// TwinCAT 3 PLC project TSG_AmazonP_LM
// ProgramVersion: 3.1.4023.0
// libraries:
//   Lynus Energy Basic, * (Lynus AG)
//   Lynus Persistent Data V1, * (Lynus AG)
//   Lynus Standards, * (Lynus AG)
//   Tc2_ModbusSrv, * (Beckhoff Automation GmbH)
//   Tc2_Standard, * (Beckhoff Automation GmbH)
//   Tc2_System, * (Beckhoff Automation GmbH)
//   Tc2_Utilities, * (Beckhoff Automation GmbH)
//   Tc3_Module, * (Beckhoff Automation GmbH)
//   TSG Communicator, * (EfficientIO)
// project tree:
//   DUTs/ FB_ECS_Alfen_NG9xx_Platform.TcPOU, FB_ECS_Alpitronic_Hypercharger.TcPOU
//   / FastTask.TcTTO, PlcTask.TcTTO
//   POUs/ prgCS1.TcPOU, prgCS2.TcPOU, prgCS3.TcPOU, prgCS4.TcPOU, prgCS5.TcPOU, prgCS6.TcPOU, prgCS7.TcPOU, prgEM.TcPOU, prgEMS.TcPOU, prgLynusCom.TcPOU, prgLynusVar.TcPOU, prgPersData.TcPOU (not stored)
// real-time tasks:
//   TASK PlcTask: cycle T#10ms, priority 8, ADS port 350
//   TASK FastTask: cycle T#5ms, priority 6, ADS port 352
// I/O:
//   DEVICE Gerät 3 (CX-BK)
//     Box 1 (CX-BK)
// variable links:
//   TSG_AmazonP_LM/TSG_AmazonP_LM Instance <-> Device 3 (CX-BK)/Box 1 (CX-BK)
//     PlcTask Inputs/prgEM.fbEM1.fbKL3403.byStateCH1 <-> Term 2 (KL3403)/Channel 1/Status
//     PlcTask Inputs/prgEM.fbEM1.fbKL3403.byStateCH2 <-> Term 2 (KL3403)/Channel 2/Status
//     PlcTask Inputs/prgEM.fbEM1.fbKL3403.byStateCH3 <-> Term 2 (KL3403)/Channel 3/Status
//     PlcTask Inputs/prgEM.fbEM2.fbKL3403.byStateCH1 <-> Term 3 (KL3403)/Channel 1/Status
//     PlcTask Inputs/prgEM.fbEM2.fbKL3403.byStateCH2 <-> Term 3 (KL3403)/Channel 2/Status
//     PlcTask Inputs/prgEM.fbEM2.fbKL3403.byStateCH3 <-> Term 3 (KL3403)/Channel 3/Status
//     PlcTask Inputs/prgEM.fbEM3.fbKL3403.byStateCH1 <-> Term 4 (KL3403)/Channel 1/Status
//     PlcTask Inputs/prgEM.fbEM3.fbKL3403.byStateCH2 <-> Term 4 (KL3403)/Channel 2/Status
//     PlcTask Inputs/prgEM.fbEM3.fbKL3403.byStateCH3 <-> Term 4 (KL3403)/Channel 3/Status
//     PlcTask Inputs/prgEM.fbEM4.fbKL3403.byStateCH1 <-> Term 5 (KL3403)/Channel 1/Status
//     PlcTask Inputs/prgEM.fbEM4.fbKL3403.byStateCH2 <-> Term 5 (KL3403)/Channel 2/Status
//     PlcTask Inputs/prgEM.fbEM4.fbKL3403.byStateCH3 <-> Term 5 (KL3403)/Channel 3/Status
//     PlcTask Inputs/prgEM.fbEM5.fbKL3403.byStateCH1 <-> Term 6 (KL3403)/Channel 1/Status
//     PlcTask Inputs/prgEM.fbEM5.fbKL3403.byStateCH2 <-> Term 6 (KL3403)/Channel 2/Status
//     PlcTask Inputs/prgEM.fbEM5.fbKL3403.byStateCH3 <-> Term 6 (KL3403)/Channel 3/Status
//     PlcTask Inputs/prgEM.fbEM6.fbKL3403.byStateCH1 <-> Term 7 (KL3403)/Channel 1/Status
//     PlcTask Inputs/prgEM.fbEM6.fbKL3403.byStateCH2 <-> Term 7 (KL3403)/Channel 2/Status
//     PlcTask Inputs/prgEM.fbEM6.fbKL3403.byStateCH3 <-> Term 7 (KL3403)/Channel 3/Status
//     PlcTask Inputs/prgEM.fbEM7.fbKL3403.byStateCH1 <-> Term 8 (KL3403)/Channel 1/Status
//     PlcTask Inputs/prgEM.fbEM7.fbKL3403.byStateCH2 <-> Term 8 (KL3403)/Channel 2/Status
//     PlcTask Inputs/prgEM.fbEM7.fbKL3403.byStateCH3 <-> Term 8 (KL3403)/Channel 3/Status
//     PlcTask Inputs/prgEM.fbEM8.fbKL3403.byStateCH1 <-> Term 9 (KL3403)/Channel 1/Status
//     PlcTask Inputs/prgEM.fbEM8.fbKL3403.byStateCH2 <-> Term 9 (KL3403)/Channel 2/Status
//     PlcTask Inputs/prgEM.fbEM8.fbKL3403.byStateCH3 <-> Term 9 (KL3403)/Channel 3/Status
//     PlcTask Inputs/prgEM.fbEM1.fbKL3403.iDataInCH1 <-> Term 2 (KL3403)/Channel 1/Daten Ein
//     PlcTask Inputs/prgEM.fbEM1.fbKL3403.iDataInCH2 <-> Term 2 (KL3403)/Channel 2/Daten Ein
//     PlcTask Inputs/prgEM.fbEM1.fbKL3403.iDataInCH3 <-> Term 2 (KL3403)/Channel 3/Daten Ein
//     PlcTask Inputs/prgEM.fbEM2.fbKL3403.iDataInCH1 <-> Term 3 (KL3403)/Channel 1/Daten Ein
//     PlcTask Inputs/prgEM.fbEM2.fbKL3403.iDataInCH2 <-> Term 3 (KL3403)/Channel 2/Daten Ein
//     PlcTask Inputs/prgEM.fbEM2.fbKL3403.iDataInCH3 <-> Term 3 (KL3403)/Channel 3/Daten Ein
//     PlcTask Inputs/prgEM.fbEM3.fbKL3403.iDataInCH1 <-> Term 4 (KL3403)/Channel 1/Daten Ein
//     PlcTask Inputs/prgEM.fbEM3.fbKL3403.iDataInCH2 <-> Term 4 (KL3403)/Channel 2/Daten Ein
//     PlcTask Inputs/prgEM.fbEM3.fbKL3403.iDataInCH3 <-> Term 4 (KL3403)/Channel 3/Daten Ein
//     PlcTask Inputs/prgEM.fbEM4.fbKL3403.iDataInCH1 <-> Term 5 (KL3403)/Channel 1/Daten Ein
//     PlcTask Inputs/prgEM.fbEM4.fbKL3403.iDataInCH2 <-> Term 5 (KL3403)/Channel 2/Daten Ein
//     PlcTask Inputs/prgEM.fbEM4.fbKL3403.iDataInCH3 <-> Term 5 (KL3403)/Channel 3/Daten Ein
//     PlcTask Inputs/prgEM.fbEM5.fbKL3403.iDataInCH1 <-> Term 6 (KL3403)/Channel 1/Daten Ein
//     PlcTask Inputs/prgEM.fbEM5.fbKL3403.iDataInCH2 <-> Term 6 (KL3403)/Channel 2/Daten Ein
//     PlcTask Inputs/prgEM.fbEM5.fbKL3403.iDataInCH3 <-> Term 6 (KL3403)/Channel 3/Daten Ein
//     PlcTask Inputs/prgEM.fbEM6.fbKL3403.iDataInCH1 <-> Term 7 (KL3403)/Channel 1/Daten Ein
//     PlcTask Inputs/prgEM.fbEM6.fbKL3403.iDataInCH2 <-> Term 7 (KL3403)/Channel 2/Daten Ein
//     PlcTask Inputs/prgEM.fbEM6.fbKL3403.iDataInCH3 <-> Term 7 (KL3403)/Channel 3/Daten Ein
//     PlcTask Inputs/prgEM.fbEM7.fbKL3403.iDataInCH1 <-> Term 8 (KL3403)/Channel 1/Daten Ein
//     PlcTask Inputs/prgEM.fbEM7.fbKL3403.iDataInCH2 <-> Term 8 (KL3403)/Channel 2/Daten Ein
//     PlcTask Inputs/prgEM.fbEM7.fbKL3403.iDataInCH3 <-> Term 8 (KL3403)/Channel 3/Daten Ein
//     PlcTask Inputs/prgEM.fbEM8.fbKL3403.iDataInCH1 <-> Term 9 (KL3403)/Channel 1/Daten Ein
//     PlcTask Inputs/prgEM.fbEM8.fbKL3403.iDataInCH2 <-> Term 9 (KL3403)/Channel 2/Daten Ein
//     PlcTask Inputs/prgEM.fbEM8.fbKL3403.iDataInCH3 <-> Term 9 (KL3403)/Channel 3/Daten Ein
//     PlcTask Inputs/prgEM.fbKBusState.uiKBusState_OUT <-> Inputs/State
//     PlcTask Outputs/prgEM.fbEM1.fbKL3403.byCntrCH1 <-> Term 2 (KL3403)/Channel 1/Kontrolle
//     PlcTask Outputs/prgEM.fbEM1.fbKL3403.byCntrCH2 <-> Term 2 (KL3403)/Channel 2/Kontrolle
//     PlcTask Outputs/prgEM.fbEM1.fbKL3403.byCntrCH3 <-> Term 2 (KL3403)/Channel 3/Kontrolle
//     PlcTask Outputs/prgEM.fbEM2.fbKL3403.byCntrCH1 <-> Term 3 (KL3403)/Channel 1/Kontrolle
//     PlcTask Outputs/prgEM.fbEM2.fbKL3403.byCntrCH2 <-> Term 3 (KL3403)/Channel 2/Kontrolle
//     PlcTask Outputs/prgEM.fbEM2.fbKL3403.byCntrCH3 <-> Term 3 (KL3403)/Channel 3/Kontrolle
//     PlcTask Outputs/prgEM.fbEM3.fbKL3403.byCntrCH1 <-> Term 4 (KL3403)/Channel 1/Kontrolle
//     PlcTask Outputs/prgEM.fbEM3.fbKL3403.byCntrCH2 <-> Term 4 (KL3403)/Channel 2/Kontrolle
//     PlcTask Outputs/prgEM.fbEM3.fbKL3403.byCntrCH3 <-> Term 4 (KL3403)/Channel 3/Kontrolle
//     PlcTask Outputs/prgEM.fbEM4.fbKL3403.byCntrCH1 <-> Term 5 (KL3403)/Channel 1/Kontrolle
//     PlcTask Outputs/prgEM.fbEM4.fbKL3403.byCntrCH2 <-> Term 5 (KL3403)/Channel 2/Kontrolle
//     PlcTask Outputs/prgEM.fbEM4.fbKL3403.byCntrCH3 <-> Term 5 (KL3403)/Channel 3/Kontrolle
//     PlcTask Outputs/prgEM.fbEM5.fbKL3403.byCntrCH1 <-> Term 6 (KL3403)/Channel 1/Kontrolle
//     PlcTask Outputs/prgEM.fbEM5.fbKL3403.byCntrCH2 <-> Term 6 (KL3403)/Channel 2/Kontrolle
//     PlcTask Outputs/prgEM.fbEM5.fbKL3403.byCntrCH3 <-> Term 6 (KL3403)/Channel 3/Kontrolle
//     PlcTask Outputs/prgEM.fbEM6.fbKL3403.byCntrCH1 <-> Term 7 (KL3403)/Channel 1/Kontrolle
//     PlcTask Outputs/prgEM.fbEM6.fbKL3403.byCntrCH2 <-> Term 7 (KL3403)/Channel 2/Kontrolle
//     PlcTask Outputs/prgEM.fbEM6.fbKL3403.byCntrCH3 <-> Term 7 (KL3403)/Channel 3/Kontrolle
//     PlcTask Outputs/prgEM.fbEM7.fbKL3403.byCntrCH1 <-> Term 8 (KL3403)/Channel 1/Kontrolle
//     PlcTask Outputs/prgEM.fbEM7.fbKL3403.byCntrCH2 <-> Term 8 (KL3403)/Channel 2/Kontrolle
//     PlcTask Outputs/prgEM.fbEM7.fbKL3403.byCntrCH3 <-> Term 8 (KL3403)/Channel 3/Kontrolle
//     PlcTask Outputs/prgEM.fbEM8.fbKL3403.byCntrCH1 <-> Term 9 (KL3403)/Channel 1/Kontrolle
//     PlcTask Outputs/prgEM.fbEM8.fbKL3403.byCntrCH2 <-> Term 9 (KL3403)/Channel 2/Kontrolle
//     PlcTask Outputs/prgEM.fbEM8.fbKL3403.byCntrCH3 <-> Term 9 (KL3403)/Channel 3/Kontrolle

CONFIGURATION TSG_AmazonP_LM
    RESOURCE PLC ON TwinCAT3
        TASK FastTask(INTERVAL := T#5ms, PRIORITY := 6);
        TASK PlcTask(INTERVAL := T#10ms, PRIORITY := 8);
        PROGRAM prgLynusVar WITH FastTask : prgLynusVar;
        PROGRAM prgEMS WITH PlcTask : prgEMS;
        PROGRAM prgEM WITH PlcTask : prgEM;
        PROGRAM prgPersData WITH PlcTask : prgPersData;
        PROGRAM prgCS2 WITH PlcTask : prgCS2;
        PROGRAM prgCS3 WITH PlcTask : prgCS3;
        PROGRAM prgCS4 WITH PlcTask : prgCS4;
        PROGRAM prgCS5 WITH PlcTask : prgCS5;
        PROGRAM prgCS6 WITH PlcTask : prgCS6;
        PROGRAM prgCS7 WITH PlcTask : prgCS7;
        PROGRAM prgCS1 WITH PlcTask : prgCS1;
        PROGRAM prgLynusCom WITH PlcTask : prgLynusCom;
    END_RESOURCE
END_CONFIGURATION

// ---- POUs/prgLynusVar.TcPOU
PROGRAM prgLynusVar
VAR
	fbVarInfo			: FB_VarInfo;
	fbRW1				: FB_ReadWrite;
	fbRW2				: FB_ReadWrite;
	fbRW3				: FB_ReadWrite;
	fbRW4				: FB_ReadWrite;
	fbRW5				: FB_ReadWrite;
	fbRW6				: FB_ReadWrite;
	fbRW7				: FB_ReadWrite;
	fbRW8				: FB_ReadWrite;
	fbRW9				: FB_ReadWrite;
	fbRW10				: FB_ReadWrite;
	
	arrCount			: ARRAY[1..10] OF UDINT;
	arrSize				: ARRAY[1..10] OF UDINT;
	
	FPError				: ARRAY[1..10] OF R_TRIG;
	arrError			: ARRAY[1..10] OF UINT;
END_VAR

fbVarInfo(
	bReadInfo:= , 
	eTMCFile:= eSelectTMCFile.eUseTMCFile, 
	eSavePositionTMCFile:= eSavePositionOnPLC.ePostionC, 
	udiCounterFoundVariables=> , 
	bError=> , 
	bBusy=> , 
	byProgress=> , 
	udiErrorCodeOut=> , 
	eErrorVarInfo_Out=> , 
	sVarWithError=> );
	
fbRW1();
fbRW2();
fbRW3();
fbRW4();
fbRW5();
fbRW6();
fbRW7();
fbRW8();
fbRW9();
fbRW10();

FPError[1](CLK:= fbRW1.bError, Q=> );
FPError[2](CLK:= fbRW2.bError, Q=> );
FPError[3](CLK:= fbRW3.bError, Q=> );
FPError[4](CLK:= fbRW4.bError, Q=> );
FPError[5](CLK:= fbRW5.bError, Q=> );
FPError[6](CLK:= fbRW6.bError, Q=> );
FPError[7](CLK:= fbRW7.bError, Q=> );
FPError[8](CLK:= fbRW8.bError, Q=> );
FPError[9](CLK:= fbRW9.bError, Q=> );
FPError[10](CLK:= fbRW10.bError, Q=> );

IF FPError[1].Q THEN arrError[1] := arrError[1] + 1; END_IF 
IF FPError[2].Q THEN arrError[2] := arrError[2] + 1; END_IF 
IF FPError[3].Q THEN arrError[3] := arrError[3] + 1; END_IF 
IF FPError[4].Q THEN arrError[4] := arrError[4] + 1; END_IF 
IF FPError[5].Q THEN arrError[5] := arrError[5] + 1; END_IF 
IF FPError[6].Q THEN arrError[6] := arrError[6] + 1; END_IF 
IF FPError[7].Q THEN arrError[7] := arrError[7] + 1; END_IF 
IF FPError[8].Q THEN arrError[8] := arrError[8] + 1; END_IF 
IF FPError[9].Q THEN arrError[9] := arrError[9] + 1; END_IF 
IF FPError[10].Q THEN arrError[10] := arrError[10] + 1; END_IF

END_PROGRAM

// ---- POUs/prgEMS.TcPOU
PROGRAM prgEMS
VAR
	fbEMS		: FB_EMS_V2;		//{#lynus.ag#()}
	
	
	//Feedback CS
	arrTarget1			: ARRAY[1..12] OF REAL;
	arrTarget2			: ARRAY[1..10] OF REAL;
	arrTarget3			: ARRAY[1..10] OF REAL;
	arrTarget4			: ARRAY[1..10] OF REAL;
	arrTarget5			: ARRAY[1..10] OF REAL;
	arrTarget6			: ARRAY[1..10] OF REAL;
	arrTarget7			: ARRAY[1..2] OF REAL;
	
	arrPower1			: ARRAY[1..12] OF LREAL;
	arrPower2			: ARRAY[1..10] OF LREAL;
	arrPower3			: ARRAY[1..10] OF LREAL;
	arrPower4			: ARRAY[1..10] OF LREAL;
	arrPower5			: ARRAY[1..10] OF LREAL;
	arrPower6			: ARRAY[1..10] OF LREAL;
	arrPower7			: ARRAY[1..2] OF LREAL;
END_VAR

fbEMS(
	bEnable:= , 
	tDelayPwrCorrectionECS:= , 
	stNrOfEM_IN_ECS:= , 
	stSizeMainFuseCS:= , 
	stSetupEMS:= , 
	eOperationMode:= , 
	eSpeedModeBackendController:= E_SpeedModeBackendController_EMS.eSlow, 
	eSpeedModeLocalController:= E_SpeedModeLocalController_EMS.eSlow, 
	bActivateHP:= , 
	bControllingState:= , 
	rHeartbeat:= , 
	rErrorWarning:= , 
	rEnergyOptReady:= , 
	rNewBattPower:= , 
	eMessageEMS=> , 
	bStateEnable=> , 
	bStateAllowChrgFromGrid=> , 
	bMissingPowerData=> , 
	bSurplusAvailable=> , 
	bSEnableMainFuseFunc=> , 
	byProgress=> , 
	uiState_OUT=> , 
	diNrOfEMS_OUT=> , 
	arrMinPrioReached=> , 
	arrMaxPrioReached=> );
	
//Feedback
arrTarget1[1] := prgCS1.fbAlfen1.stDataECS.rTargetPower;
arrTarget1[2] := prgCS1.fbAlfen2.stDataECS.rTargetPower;
arrTarget1[3] := prgCS1.fbAlfen3.stDataECS.rTargetPower;
arrTarget1[4] := prgCS1.fbAlfen4.stDataECS.rTargetPower;
arrTarget1[5] := prgCS1.fbAlfen5.stDataECS.rTargetPower;
arrTarget1[6] := prgCS1.fbAlfen6.stDataECS.rTargetPower;
arrTarget1[7] := prgCS1.fbAlfen7.stDataECS.rTargetPower;
arrTarget1[8] := prgCS1.fbAlfen8.stDataECS.rTargetPower;
arrTarget1[9] := prgCS1.fbAlfen9.stDataECS.rTargetPower;
arrTarget1[10] := prgCS1.fbAlfen10.stDataECS.rTargetPower;
arrTarget1[11] := prgCS1.fbApliT_1.stDataECS.rTargetPower;
arrTarget1[12] := prgCS1.fbApliT_2.stDataECS.rTargetPower;

arrTarget2[1] := prgCS2.fbAlfen1.stDataECS.rTargetPower;
arrTarget2[2] := prgCS2.fbAlfen2.stDataECS.rTargetPower;
arrTarget2[3] := prgCS2.fbAlfen3.stDataECS.rTargetPower;
arrTarget2[4] := prgCS2.fbAlfen4.stDataECS.rTargetPower;
arrTarget2[5] := prgCS2.fbAlfen5.stDataECS.rTargetPower;
arrTarget2[6] := prgCS2.fbAlfen6.stDataECS.rTargetPower;
arrTarget2[7] := prgCS2.fbAlfen7.stDataECS.rTargetPower;
arrTarget2[8] := prgCS2.fbAlfen8.stDataECS.rTargetPower;
arrTarget2[9] := prgCS2.fbAlfen9.stDataECS.rTargetPower;
arrTarget2[10] := prgCS2.fbAlfen10.stDataECS.rTargetPower;

arrTarget3[1] := prgCS3.fbAlfen1.stDataECS.rTargetPower;
arrTarget3[2] := prgCS3.fbAlfen2.stDataECS.rTargetPower;
arrTarget3[3] := prgCS3.fbAlfen3.stDataECS.rTargetPower;
arrTarget3[4] := prgCS3.fbAlfen4.stDataECS.rTargetPower;
arrTarget3[5] := prgCS3.fbAlfen5.stDataECS.rTargetPower;
arrTarget3[6] := prgCS3.fbAlfen6.stDataECS.rTargetPower;
arrTarget3[7] := prgCS3.fbAlfen7.stDataECS.rTargetPower;
arrTarget3[8] := prgCS3.fbAlfen8.stDataECS.rTargetPower;
arrTarget3[9] := prgCS3.fbAlfen9.stDataECS.rTargetPower;
arrTarget3[10] := prgCS3.fbAlfen10.stDataECS.rTargetPower;

arrTarget4[1] := prgCS4.fbAlfen1.stDataECS.rTargetPower;
arrTarget4[2] := prgCS4.fbAlfen2.stDataECS.rTargetPower;
arrTarget4[3] := prgCS4.fbAlfen3.stDataECS.rTargetPower;
arrTarget4[4] := prgCS4.fbAlfen4.stDataECS.rTargetPower;
arrTarget4[5] := prgCS4.fbAlfen5.stDataECS.rTargetPower;
arrTarget4[6] := prgCS4.fbAlfen6.stDataECS.rTargetPower;
arrTarget4[7] := prgCS4.fbAlfen7.stDataECS.rTargetPower;
arrTarget4[8] := prgCS4.fbAlfen8.stDataECS.rTargetPower;
arrTarget4[9] := prgCS4.fbAlfen9.stDataECS.rTargetPower;
arrTarget4[10] := prgCS4.fbAlfen10.stDataECS.rTargetPower;

arrTarget5[1] := prgCS5.fbAlfen1.stDataECS.rTargetPower;
arrTarget5[2] := prgCS5.fbAlfen2.stDataECS.rTargetPower;
arrTarget5[3] := prgCS5.fbAlfen3.stDataECS.rTargetPower;
arrTarget5[4] := prgCS5.fbAlfen4.stDataECS.rTargetPower;
arrTarget5[5] := prgCS5.fbAlfen5.stDataECS.rTargetPower;
arrTarget5[6] := prgCS5.fbAlfen6.stDataECS.rTargetPower;
arrTarget5[7] := prgCS5.fbAlfen7.stDataECS.rTargetPower;
arrTarget5[8] := prgCS5.fbAlfen8.stDataECS.rTargetPower;
arrTarget5[9] := prgCS5.fbAlfen9.stDataECS.rTargetPower;
arrTarget5[10] := prgCS5.fbAlfen10.stDataECS.rTargetPower;

arrTarget6[1] := prgCS6.fbAlfen1.stDataECS.rTargetPower;
arrTarget6[2] := prgCS6.fbAlfen2.stDataECS.rTargetPower;
arrTarget6[3] := prgCS6.fbAlfen3.stDataECS.rTargetPower;
arrTarget6[4] := prgCS6.fbAlfen4.stDataECS.rTargetPower;
arrTarget6[5] := prgCS6.fbAlfen5.stDataECS.rTargetPower;
arrTarget6[6] := prgCS6.fbAlfen6.stDataECS.rTargetPower;
arrTarget6[7] := prgCS6.fbAlfen7.stDataECS.rTargetPower;
arrTarget6[8] := prgCS6.fbAlfen8.stDataECS.rTargetPower;
arrTarget6[9] := prgCS6.fbAlfen9.stDataECS.rTargetPower;
arrTarget6[10] := prgCS6.fbAlfen10.stDataECS.rTargetPower;

arrTarget7[1] := prgCS7.fbAlfen1.stDataECS.rTargetPower;
arrTarget7[2] := prgCS7.fbAlfen2.stDataECS.rTargetPower;

//Power
arrPower1[1] := prgCS1.fbAlfen1.stDataECS.lrTotalPower;
arrPower1[2] := prgCS1.fbAlfen2.stDataECS.lrTotalPower;
arrPower1[3] := prgCS1.fbAlfen3.stDataECS.lrTotalPower;
arrPower1[4] := prgCS1.fbAlfen4.stDataECS.lrTotalPower;
arrPower1[5] := prgCS1.fbAlfen5.stDataECS.lrTotalPower;
arrPower1[6] := prgCS1.fbAlfen6.stDataECS.lrTotalPower;
arrPower1[7] := prgCS1.fbAlfen7.stDataECS.lrTotalPower;
arrPower1[8] := prgCS1.fbAlfen8.stDataECS.lrTotalPower;
arrPower1[9] := prgCS1.fbAlfen9.stDataECS.lrTotalPower;
arrPower1[10] := prgCS1.fbAlfen10.stDataECS.lrTotalPower;
arrPower1[11] := prgCS1.fbApliT_1.stDataECS.lrTotalPower;
arrPower1[12] := prgCS1.fbApliT_2.stDataECS.lrTotalPower;

arrPower2[1] := prgCS2.fbAlfen1.stDataECS.lrTotalPower;
arrPower2[2] := prgCS2.fbAlfen2.stDataECS.lrTotalPower;
arrPower2[3] := prgCS2.fbAlfen3.stDataECS.lrTotalPower;
arrPower2[4] := prgCS2.fbAlfen4.stDataECS.lrTotalPower;
arrPower2[5] := prgCS2.fbAlfen5.stDataECS.lrTotalPower;
arrPower2[6] := prgCS2.fbAlfen6.stDataECS.lrTotalPower;
arrPower2[7] := prgCS2.fbAlfen7.stDataECS.lrTotalPower;
arrPower2[8] := prgCS2.fbAlfen8.stDataECS.lrTotalPower;
arrPower2[9] := prgCS2.fbAlfen9.stDataECS.lrTotalPower;
arrPower2[10] := prgCS2.fbAlfen10.stDataECS.lrTotalPower;

arrPower3[1] := prgCS3.fbAlfen1.stDataECS.lrTotalPower;
arrPower3[2] := prgCS3.fbAlfen2.stDataECS.lrTotalPower;
arrPower3[3] := prgCS3.fbAlfen3.stDataECS.lrTotalPower;
arrPower3[4] := prgCS3.fbAlfen4.stDataECS.lrTotalPower;
arrPower3[5] := prgCS3.fbAlfen5.stDataECS.lrTotalPower;
arrPower3[6] := prgCS3.fbAlfen6.stDataECS.lrTotalPower;
arrPower3[7] := prgCS3.fbAlfen7.stDataECS.lrTotalPower;
arrPower3[8] := prgCS3.fbAlfen8.stDataECS.lrTotalPower;
arrPower3[9] := prgCS3.fbAlfen9.stDataECS.lrTotalPower;
arrPower3[10] := prgCS3.fbAlfen10.stDataECS.lrTotalPower;

arrPower4[1] := prgCS4.fbAlfen1.stDataECS.lrTotalPower;
arrPower4[2] := prgCS4.fbAlfen2.stDataECS.lrTotalPower;
arrPower4[3] := prgCS4.fbAlfen3.stDataECS.lrTotalPower;
arrPower4[4] := prgCS4.fbAlfen4.stDataECS.lrTotalPower;
arrPower4[5] := prgCS4.fbAlfen5.stDataECS.lrTotalPower;
arrPower4[6] := prgCS4.fbAlfen6.stDataECS.lrTotalPower;
arrPower4[7] := prgCS4.fbAlfen7.stDataECS.lrTotalPower;
arrPower4[8] := prgCS4.fbAlfen8.stDataECS.lrTotalPower;
arrPower4[9] := prgCS4.fbAlfen9.stDataECS.lrTotalPower;
arrPower4[10] := prgCS4.fbAlfen10.stDataECS.lrTotalPower;

arrPower5[1] := prgCS5.fbAlfen1.stDataECS.lrTotalPower;
arrPower5[2] := prgCS5.fbAlfen2.stDataECS.lrTotalPower;
arrPower5[3] := prgCS5.fbAlfen3.stDataECS.lrTotalPower;
arrPower5[4] := prgCS5.fbAlfen4.stDataECS.lrTotalPower;
arrPower5[5] := prgCS5.fbAlfen5.stDataECS.lrTotalPower;
arrPower5[6] := prgCS5.fbAlfen6.stDataECS.lrTotalPower;
arrPower5[7] := prgCS5.fbAlfen7.stDataECS.lrTotalPower;
arrPower5[8] := prgCS5.fbAlfen8.stDataECS.lrTotalPower;
arrPower5[9] := prgCS5.fbAlfen9.stDataECS.lrTotalPower;
arrPower5[10] := prgCS5.fbAlfen10.stDataECS.lrTotalPower;

arrPower6[1] := prgCS6.fbAlfen1.stDataECS.lrTotalPower;
arrPower6[2] := prgCS6.fbAlfen2.stDataECS.lrTotalPower;
arrPower6[3] := prgCS6.fbAlfen3.stDataECS.lrTotalPower;
arrPower6[4] := prgCS6.fbAlfen4.stDataECS.lrTotalPower;
arrPower6[5] := prgCS6.fbAlfen5.stDataECS.lrTotalPower;
arrPower6[6] := prgCS6.fbAlfen6.stDataECS.lrTotalPower;
arrPower6[7] := prgCS6.fbAlfen7.stDataECS.lrTotalPower;
arrPower6[8] := prgCS6.fbAlfen8.stDataECS.lrTotalPower;
arrPower6[9] := prgCS6.fbAlfen9.stDataECS.lrTotalPower;
arrPower6[10] := prgCS6.fbAlfen10.stDataECS.lrTotalPower;

arrPower7[1] := prgCS7.fbAlfen1.stDataECS.lrTotalPower;
arrPower7[2] := prgCS7.fbAlfen2.stDataECS.lrTotalPower;

END_PROGRAM

// ---- POUs/prgCS1.TcPOU
PROGRAM prgCS1
VAR
	fbAlfen1					: FB_ECS_Alfen_NG9xx_Platform;						//{#lynus.ag#()}
	fbAlfen2					: FB_ECS_Alfen_NG9xx_Platform;						//{#lynus.ag#()}
	fbAlfen3					: FB_ECS_Alfen_NG9xx_Platform;						//{#lynus.ag#()}
	fbAlfen4					: FB_ECS_Alfen_NG9xx_Platform;						//{#lynus.ag#()}
	fbAlfen5					: FB_ECS_Alfen_NG9xx_Platform;						//{#lynus.ag#()}
	fbAlfen6					: FB_ECS_Alfen_NG9xx_Platform;						//{#lynus.ag#()}
	fbAlfen7					: FB_ECS_Alfen_NG9xx_Platform;						//{#lynus.ag#()}
	fbAlfen8					: FB_ECS_Alfen_NG9xx_Platform;						//{#lynus.ag#()}
	fbAlfen9					: FB_ECS_Alfen_NG9xx_Platform;						//{#lynus.ag#()}
	fbAlfen10					: FB_ECS_Alfen_NG9xx_Platform;						//{#lynus.ag#()}
	fbApliT_1					: FB_ECS_Alpitronic_Hypercharger;					//{#lynus.ag#()}
	fbApliT_2					: FB_ECS_Alpitronic_Hypercharger;					//{#lynus.ag#()}
	
	bSManualyOn_UV1_1			: BOOL;												//{#lynus.ag#()}
	bySManualyTargetPowerUV1_1	: BYTE;												//{#lynus.ag#()}
	byErrorWarningUV1_1			: BYTE;												//{#lynus.ag#()}
	rChargingTimeInMinUV1_1		: REAL;												//{#lynus.ag#()}
	lrPowerUV1_1				: LREAL;											//{#lynus.ag#()}
	wStateUV1_1					: WORD;												//{#lynus.ag#()}
	lrEnergySessionUV1_1		: LREAL;											//{#lynus.ag#()}
	lrTotalEnergyUV1_1			: LREAL;											//{#lynus.ag#()}
	
	bSManualyOn_UV1_2			: BOOL;												//{#lynus.ag#()}
	bySManualyTargetPowerUV1_2	: BYTE;												//{#lynus.ag#()}
	byErrorWarningUV1_2			: BYTE;												//{#lynus.ag#()}
	rChargingTimeInMinUV1_2		: REAL;												//{#lynus.ag#()}
	lrPowerUV1_2				: LREAL;											//{#lynus.ag#()}
	wStateUV1_2					: WORD;												//{#lynus.ag#()}
	lrEnergySessionUV1_2		: LREAL;											//{#lynus.ag#()}
	lrTotalEnergyUV1_2			: LREAL;											//{#lynus.ag#()}
	
	bSManualyOn_UV1_3			: BOOL;												//{#lynus.ag#()}
	bySManualyTargetPowerUV1_3	: BYTE;												//{#lynus.ag#()}
	byErrorWarningUV1_3			: BYTE;												//{#lynus.ag#()}
	rChargingTimeInMinUV1_3		: REAL;												//{#lynus.ag#()}
	lrPowerUV1_3				: LREAL;											//{#lynus.ag#()}
	wStateUV1_3					: WORD;												//{#lynus.ag#()}
	lrEnergySessionUV1_3		: LREAL;											//{#lynus.ag#()}
	lrTotalEnergyUV1_3			: LREAL;											//{#lynus.ag#()}
	
	bSManualyOn_UV1_4			: BOOL;												//{#lynus.ag#()}
	bySManualyTargetPowerUV1_4	: BYTE;												//{#lynus.ag#()}
	byErrorWarningUV1_4			: BYTE;												//{#lynus.ag#()}
	rChargingTimeInMinUV1_4		: REAL;												//{#lynus.ag#()}
	lrPowerUV1_4				: LREAL;											//{#lynus.ag#()}
	wStateUV1_4					: WORD;												//{#lynus.ag#()}
	lrEnergySessionUV1_4		: LREAL;											//{#lynus.ag#()}
	lrTotalEnergyUV1_4			: LREAL;											//{#lynus.ag#()}
	
	bSManualyOn_UV1_5			: BOOL;												//{#lynus.ag#()}
	bySManualyTargetPowerUV1_5	: BYTE;												//{#lynus.ag#()}
	byErrorWarningUV1_5			: BYTE;												//{#lynus.ag#()}
	rChargingTimeInMinUV1_5		: REAL;												//{#lynus.ag#()}
	lrPowerUV1_5				: LREAL;											//{#lynus.ag#()}
	wStateUV1_5					: WORD;												//{#lynus.ag#()}
	lrEnergySessionUV1_5		: LREAL;											//{#lynus.ag#()}
	lrTotalEnergyUV1_5			: LREAL;											//{#lynus.ag#()}
	
	bSManualyOn_UV1_6			: BOOL;												//{#lynus.ag#()}
	bySManualyTargetPowerUV1_6	: BYTE;												//{#lynus.ag#()}
	byErrorWarningUV1_6			: BYTE;												//{#lynus.ag#()}
	rChargingTimeInMinUV1_6		: REAL;												//{#lynus.ag#()}
	lrPowerUV1_6				: LREAL;											//{#lynus.ag#()}
	wStateUV1_6					: WORD;												//{#lynus.ag#()}
	lrEnergySessionUV1_6		: LREAL;											//{#lynus.ag#()}
	lrTotalEnergyUV1_6			: LREAL;											//{#lynus.ag#()}
	
	bSManualyOn_UV1_7			: BOOL;												//{#lynus.ag#()}
	bySManualyTargetPowerUV1_7	: BYTE;												//{#lynus.ag#()}
	byErrorWarningUV1_7			: BYTE;												//{#lynus.ag#()}
	rChargingTimeInMinUV1_7		: REAL;												//{#lynus.ag#()}
	lrPowerUV1_7				: LREAL;											//{#lynus.ag#()}
	wStateUV1_7					: WORD;												//{#lynus.ag#()}
	lrEnergySessionUV1_7		: LREAL;											//{#lynus.ag#()}
	lrTotalEnergyUV1_7			: LREAL;											//{#lynus.ag#()}
	
	bSManualyOn_UV1_8			: BOOL;												//{#lynus.ag#()}
	bySManualyTargetPowerUV1_8	: BYTE;												//{#lynus.ag#()}
	byErrorWarningUV1_8			: BYTE;												//{#lynus.ag#()}
	rChargingTimeInMinUV1_8		: REAL;												//{#lynus.ag#()}
	lrPowerUV1_8				: LREAL;											//{#lynus.ag#()}
	wStateUV1_8					: WORD;												//{#lynus.ag#()}
	lrEnergySessionUV1_8		: LREAL;											//{#lynus.ag#()}
	lrTotalEnergyUV1_8			: LREAL;											//{#lynus.ag#()}
	
	bSManualyOn_UV1_9			: BOOL;												//{#lynus.ag#()}
	bySManualyTargetPowerUV1_9	: BYTE;												//{#lynus.ag#()}
	byErrorWarningUV1_9			: BYTE;												//{#lynus.ag#()}
	rChargingTimeInMinUV1_9		: REAL;												//{#lynus.ag#()}
	lrPowerUV1_9				: LREAL;											//{#lynus.ag#()}
	wStateUV1_9					: WORD;												//{#lynus.ag#()}
	lrEnergySessionUV1_9		: LREAL;											//{#lynus.ag#()}
	lrTotalEnergyUV1_9			: LREAL;											//{#lynus.ag#()}
	
	bSManualyOn_UV1_10			: BOOL;												//{#lynus.ag#()}
	bySManualyTargetPowerUV1_10	: BYTE;												//{#lynus.ag#()}
	byErrorWarningUV1_10		: BYTE;												//{#lynus.ag#()}
	rChargingTimeInMinUV1_10	: REAL;												//{#lynus.ag#()}
	lrPowerUV1_10				: LREAL;											//{#lynus.ag#()}
	wStateUV1_10				: WORD;												//{#lynus.ag#()}
	lrEnergySessionUV1_10		: LREAL;											//{#lynus.ag#()}
	lrTotalEnergyUV1_10			: LREAL;											//{#lynus.ag#()}
	
	bSManualyOn_DC_1			: BOOL;												//{#lynus.ag#()}
	bySManualyTargetPowerDC_1	: BYTE;												//{#lynus.ag#()}
	byErrorWarningDC_1			: BYTE;												//{#lynus.ag#()}
	lrPowerTotalDC1				: LREAL;											//{#lynus.ag#()}
	lrPowerDC1_S1				: LREAL;											//{#lynus.ag#()}
	lrPowerDC1_S2				: LREAL;											//{#lynus.ag#()}
	rChargingTimeInMinDC1_S1	: REAL;												//{#lynus.ag#()}
	rChargingTimeInMinDC1_S2	: REAL;												//{#lynus.ag#()}
	dwSOCCarDC1_S1				: DWORD;											//{#lynus.ag#()}
	dwSOCCarDC1_S2				: DWORD;											//{#lynus.ag#()}
	wStateDC1_S1				: WORD;												//{#lynus.ag#()}
	wStateDC1_S2				: WORD;												//{#lynus.ag#()}
	lrEnergySessionDC1_S1		: LREAL;											//{#lynus.ag#()}
	lrEnergySessionDC1_S2		: LREAL;											//{#lynus.ag#()}
	lrTotalEnergyDC1			: LREAL;											//{#lynus.ag#()}
	
	bSManualyOn_DC_2			: BOOL;												//{#lynus.ag#()}
	bySManualyTargetPowerDC_2	: BYTE;												//{#lynus.ag#()}
	byErrorWarningDC_2			: BYTE;												//{#lynus.ag#()}
	lrPowerTotalDC2				: LREAL;											//{#lynus.ag#()}
	lrPowerDC2_S1				: LREAL;											//{#lynus.ag#()}
	lrPowerDC2_S2				: LREAL;											//{#lynus.ag#()}
	rChargingTimeInMinDC2_S1	: REAL;												//{#lynus.ag#()}
	rChargingTimeInMinDC2_S2	: REAL;												//{#lynus.ag#()}
	dwSOCCarDC2_S1				: DWORD;											//{#lynus.ag#()}
	dwSOCCarDC2_S2				: DWORD;											//{#lynus.ag#()}
	wStateDC2_S1				: WORD;												//{#lynus.ag#()}
	wStateDC2_S2				: WORD;												//{#lynus.ag#()}
	lrEnergySessionDC2_S1		: LREAL;											//{#lynus.ag#()}
	lrEnergySessionDC2_S2		: LREAL;											//{#lynus.ag#()}
	lrTotalEnergyDC2			: LREAL;											//{#lynus.ag#()}
END_VAR
VAR PERSISTENT
	bManualyOnUV1_1				: BOOL;												//{#lynus.ag#()}
	byManualyTargetPowerUV1_1	: BYTE;												//{#lynus.ag#()}
	
	bManualyOnUV1_2				: BOOL;												//{#lynus.ag#()}
	byManualyTargetPowerUV1_2	: BYTE;												//{#lynus.ag#()}
	
	bManualyOnUV1_3				: BOOL;												//{#lynus.ag#()}
	byManualyTargetPowerUV1_3	: BYTE;												//{#lynus.ag#()}
	
	bManualyOnUV1_4				: BOOL;												//{#lynus.ag#()}
	byManualyTargetPowerUV1_4	: BYTE;												//{#lynus.ag#()}
	
	bManualyOnUV1_5				: BOOL;												//{#lynus.ag#()}
	byManualyTargetPowerUV1_5	: BYTE;												//{#lynus.ag#()}
	
	bManualyOnUV1_6				: BOOL;												//{#lynus.ag#()}
	byManualyTargetPowerUV1_6	: BYTE;												//{#lynus.ag#()}
	
	bManualyOnUV1_7				: BOOL;												//{#lynus.ag#()}
	byManualyTargetPowerUV1_7	: BYTE;												//{#lynus.ag#()}
	
	bManualyOnUV1_8				: BOOL;												//{#lynus.ag#()}
	byManualyTargetPowerUV1_8	: BYTE;												//{#lynus.ag#()}
	
	bManualyOnUV1_9				: BOOL;												//{#lynus.ag#()}
	byManualyTargetPowerUV1_9	: BYTE;												//{#lynus.ag#()}
	
	bManualyOnUV1_10			: BOOL;												//{#lynus.ag#()}
	byManualyTargetPowerUV1_10	: BYTE;												//{#lynus.ag#()}
	
	bManualyOnDC_1				: BOOL;												//{#lynus.ag#()}
	byManualyTargetPowerDC_1	: BYTE;												//{#lynus.ag#()}
	
	bManualyOnDC_2				: BOOL;												//{#lynus.ag#()}
	byManualyTargetPowerDC_2	: BYTE;												//{#lynus.ag#()}
END_VAR

(*---------------------------------------------CS1-----------------------------------------------------------*)

//Manual Power
fbAlfen1.stSetupECS.bManualyOn := bManualyOnUV1_1;
	fbAlfen1.stSetupECS.byManualyTargetPower := byManualyTargetPowerUV1_1;

fbAlfen1(
	bEnable:= , 
	bPowerDataInvers:= , 
	byElectricFuseLine:= , 
	byUnitID_Socket1:= 1, 
	byUnitID_Socket2:= , 
	byNumberOfSockets:= 1, 
	byNumberOfConnectionWire:= 1, 
	diNrOfEMS_IN:= prgEMS.fbEMS.diNrOfEMS_OUT, 
	diNrOfEM_IN_CS:= , 
	sIPAdress:= '192.168.1.123', 
	stSetupECS:= , 
	stDataECS=> , 
	diNrOfECS_OUT=> );

bSManualyOn_UV1_1 := fbAlfen1.stDataECS.bSManualyOn;
	bySManualyTargetPowerUV1_1 := fbAlfen1.stDataECS.bySManualyTargetPower;
		byErrorWarningUV1_1 := fbAlfen1.stDataECS.byErrorWarning;	
			rChargingTimeInMinUV1_1 := fbAlfen1.stDataECS.arrChargingTimeInMin[1];
				lrPowerUV1_1 := fbAlfen1.stDataECS.lrTotalPower;	
					wStateUV1_1 := fbAlfen1.stDataECS.arrSocketStateECS[1];
						lrEnergySessionUV1_1 := fbAlfen1.stDataECS.arrSocketEnergySession[1];
							lrTotalEnergyUV1_1 := fbAlfen1.stDataECS.lrTotalCounterEnergy_Consumption;		
	
(*---------------------------------------------CS2-----------------------------------------------------------*)
	
//Manual Power
fbAlfen2.stSetupECS.bManualyOn := bManualyOnUV1_2;
	fbAlfen2.stSetupECS.byManualyTargetPower := byManualyTargetPowerUV1_2;
	
fbAlfen2(
	bEnable:= , 
	bPowerDataInvers:= , 
	byElectricFuseLine:= , 
	byUnitID_Socket1:= 1, 
	byUnitID_Socket2:= , 
	byNumberOfSockets:= 1, 
	byNumberOfConnectionWire:= 1, 
	diNrOfEMS_IN:= prgEMS.fbEMS.diNrOfEMS_OUT, 
	diNrOfEM_IN_CS:= , 
	sIPAdress:= '192.168.1.111', 
	stSetupECS:= , 
	stDataECS=> , 
	diNrOfECS_OUT=> );

bSManualyOn_UV1_2 := fbAlfen2.stDataECS.bSManualyOn;
	bySManualyTargetPowerUV1_2 := fbAlfen2.stDataECS.bySManualyTargetPower;	
		byErrorWarningUV1_2 := fbAlfen2.stDataECS.byErrorWarning;
			rChargingTimeInMinUV1_2 := fbAlfen2.stDataECS.arrChargingTimeInMin[1];;
				lrPowerUV1_2 := fbAlfen2.stDataECS.lrTotalPower;	
					wStateUV1_2 := fbAlfen2.stDataECS.arrSocketStateECS[1];
						lrEnergySessionUV1_2 := fbAlfen2.stDataECS.arrSocketEnergySession[1];
							lrTotalEnergyUV1_2 := fbAlfen2.stDataECS.lrTotalCounterEnergy_Consumption;
	
(*---------------------------------------------CS3-----------------------------------------------------------*)	
	
//Manual Power
fbAlfen3.stSetupECS.bManualyOn := bManualyOnUV1_3;
	fbAlfen3.stSetupECS.byManualyTargetPower := byManualyTargetPowerUV1_3;
	
fbAlfen3(
	bEnable:= , 
	bPowerDataInvers:= , 
	byElectricFuseLine:= , 
	byUnitID_Socket1:= 1, 
	byUnitID_Socket2:= , 
	byNumberOfSockets:= 1, 
	byNumberOfConnectionWire:= 1, 
	diNrOfEMS_IN:= prgEMS.fbEMS.diNrOfEMS_OUT, 
	diNrOfEM_IN_CS:= , 
	sIPAdress:= '192.168.1.213',  
	stSetupECS:= , 
	stDataECS=> , 
	diNrOfECS_OUT=> );

bSManualyOn_UV1_3 := fbAlfen3.stDataECS.bSManualyOn;
	bySManualyTargetPowerUV1_3 := fbAlfen3.stDataECS.bySManualyTargetPower;
		byErrorWarningUV1_3 := fbAlfen3.stDataECS.byErrorWarning;
			rChargingTimeInMinUV1_3 := fbAlfen3.stDataECS.arrChargingTimeInMin[1];	
				lrPowerUV1_3 := fbAlfen3.stDataECS.lrTotalPower;	
					wStateUV1_3 := fbAlfen3.stDataECS.arrSocketStateECS[1];
						lrEnergySessionUV1_3 := fbAlfen3.stDataECS.arrSocketEnergySession[1];
							lrTotalEnergyUV1_3 := fbAlfen3.stDataECS.lrTotalCounterEnergy_Consumption;
	
(*---------------------------------------------CS4-----------------------------------------------------------*)	
	
//Manual Power
fbAlfen4.stSetupECS.bManualyOn := bManualyOnUV1_4;
	fbAlfen4.stSetupECS.byManualyTargetPower := byManualyTargetPowerUV1_4;
	
fbAlfen4(
	bEnable:= , 
	bPowerDataInvers:= , 
	byElectricFuseLine:= , 
	byUnitID_Socket1:= 1, 
	byUnitID_Socket2:= , 
	byNumberOfSockets:= 1, 
	byNumberOfConnectionWire:= 1, 
	diNrOfEMS_IN:= prgEMS.fbEMS.diNrOfEMS_OUT, 
	diNrOfEM_IN_CS:= , 
	sIPAdress:= '192.168.1.144',  
	stSetupECS:= , 
	stDataECS=> , 
	diNrOfECS_OUT=> );

bSManualyOn_UV1_4 := fbAlfen4.stDataECS.bSManualyOn;
	bySManualyTargetPowerUV1_4 := fbAlfen4.stDataECS.bySManualyTargetPower;	
		byErrorWarningUV1_4 := fbAlfen4.stDataECS.byErrorWarning;
			rChargingTimeInMinUV1_4 := fbAlfen4.stDataECS.arrChargingTimeInMin[1];
				lrPowerUV1_4 := fbAlfen4.stDataECS.lrTotalPower;	
					wStateUV1_4 := fbAlfen4.stDataECS.arrSocketStateECS[1];
						lrEnergySessionUV1_4 := fbAlfen4.stDataECS.arrSocketEnergySession[1];
							lrTotalEnergyUV1_4 := fbAlfen4.stDataECS.lrTotalCounterEnergy_Consumption;
	
(*---------------------------------------------CS5-----------------------------------------------------------*)	
	
//Manual Power
fbAlfen5.stSetupECS.bManualyOn := bManualyOnUV1_5;
	fbAlfen5.stSetupECS.byManualyTargetPower := byManualyTargetPowerUV1_5;
	
fbAlfen5(
	bEnable:= , 
	bPowerDataInvers:= , 
	byElectricFuseLine:= , 
	byUnitID_Socket1:= 1, 
	byUnitID_Socket2:= , 
	byNumberOfSockets:= 1, 
	byNumberOfConnectionWire:= 1, 
	diNrOfEMS_IN:= prgEMS.fbEMS.diNrOfEMS_OUT, 
	diNrOfEM_IN_CS:= , 
	sIPAdress:= '192.168.1.178',  
	stSetupECS:= , 
	stDataECS=> , 
	diNrOfECS_OUT=> );

bSManualyOn_UV1_5 := fbAlfen5.stDataECS.bSManualyOn;
	bySManualyTargetPowerUV1_5 := fbAlfen5.stDataECS.bySManualyTargetPower;
		byErrorWarningUV1_5 := fbAlfen5.stDataECS.byErrorWarning;
			rChargingTimeInMinUV1_5 := fbAlfen5.stDataECS.arrChargingTimeInMin[1];
				lrPowerUV1_5 := fbAlfen5.stDataECS.lrTotalPower;	
					wStateUV1_5 := fbAlfen5.stDataECS.arrSocketStateECS[1];
						lrEnergySessionUV1_5 := fbAlfen5.stDataECS.arrSocketEnergySession[1];
							lrTotalEnergyUV1_5 := fbAlfen5.stDataECS.lrTotalCounterEnergy_Consumption;	
	
(*---------------------------------------------CS6-----------------------------------------------------------*)	
	
//Manual Power
fbAlfen6.stSetupECS.bManualyOn := bManualyOnUV1_6;
	fbAlfen6.stSetupECS.byManualyTargetPower := byManualyTargetPowerUV1_6;
	
fbAlfen6(
	bEnable:= , 
	bPowerDataInvers:= , 
	byElectricFuseLine:= , 
	byUnitID_Socket1:= 1, 
	byUnitID_Socket2:= , 
	byNumberOfSockets:= 1, 
	byNumberOfConnectionWire:= 1, 
	diNrOfEMS_IN:= prgEMS.fbEMS.diNrOfEMS_OUT, 
	diNrOfEM_IN_CS:= , 
	sIPAdress:= '192.168.1.161',  
	stSetupECS:= , 
	stDataECS=> , 
	diNrOfECS_OUT=> );

bSManualyOn_UV1_6 := fbAlfen6.stDataECS.bSManualyOn;
	bySManualyTargetPowerUV1_6 := fbAlfen6.stDataECS.bySManualyTargetPower;	
		byErrorWarningUV1_6 := fbAlfen6.stDataECS.byErrorWarning;
			rChargingTimeInMinUV1_6 := fbAlfen6.stDataECS.arrChargingTimeInMin[1];
				lrPowerUV1_6 := fbAlfen6.stDataECS.lrTotalPower;	
					wStateUV1_6 := fbAlfen6.stDataECS.arrSocketStateECS[1];
						lrEnergySessionUV1_6 := fbAlfen6.stDataECS.arrSocketEnergySession[1];
							lrTotalEnergyUV1_6 := fbAlfen6.stDataECS.lrTotalCounterEnergy_Consumption;
	
(*---------------------------------------------CS7-----------------------------------------------------------*)	
	
//Manual Power
fbAlfen7.stSetupECS.bManualyOn := bManualyOnUV1_7;
	fbAlfen7.stSetupECS.byManualyTargetPower := byManualyTargetPowerUV1_7;
	
fbAlfen7(
	bEnable:= , 
	bPowerDataInvers:= , 
	byElectricFuseLine:= , 
	byUnitID_Socket1:= 1, 
	byUnitID_Socket2:= , 
	byNumberOfSockets:= 1, 
	byNumberOfConnectionWire:= 1, 
	diNrOfEMS_IN:= prgEMS.fbEMS.diNrOfEMS_OUT, 
	diNrOfEM_IN_CS:= , 
	sIPAdress:= '192.168.1.241',  
	stSetupECS:= , 
	stDataECS=> , 
	diNrOfECS_OUT=> );

bSManualyOn_UV1_7 := fbAlfen7.stDataECS.bSManualyOn;
	bySManualyTargetPowerUV1_7 := fbAlfen7.stDataECS.bySManualyTargetPower;	
		byErrorWarningUV1_7 := fbAlfen7.stDataECS.byErrorWarning;
			rChargingTimeInMinUV1_7 := fbAlfen7.stDataECS.arrChargingTimeInMin[1];
				lrPowerUV1_7 := fbAlfen7.stDataECS.lrTotalPower;	
					wStateUV1_7 := fbAlfen7.stDataECS.arrSocketStateECS[1];
						lrEnergySessionUV1_7 := fbAlfen7.stDataECS.arrSocketEnergySession[1];
							lrTotalEnergyUV1_7 := fbAlfen7.stDataECS.lrTotalCounterEnergy_Consumption;
	
(*---------------------------------------------CS8-----------------------------------------------------------*)	
	
//Manual Power
fbAlfen8.stSetupECS.bManualyOn := bManualyOnUV1_8;
	fbAlfen8.stSetupECS.byManualyTargetPower := byManualyTargetPowerUV1_8;
	
fbAlfen8(
	bEnable:= , 
	bPowerDataInvers:= , 
	byElectricFuseLine:= , 
	byUnitID_Socket1:= 1, 
	byUnitID_Socket2:= , 
	byNumberOfSockets:= 1, 
	byNumberOfConnectionWire:= 1, 
	diNrOfEMS_IN:= prgEMS.fbEMS.diNrOfEMS_OUT, 
	diNrOfEM_IN_CS:= , 
	sIPAdress:= '192.168.1.124',  
	stSetupECS:= , 
	stDataECS=> , 
	diNrOfECS_OUT=> );

bSManualyOn_UV1_8 := fbAlfen8.stDataECS.bSManualyOn;
	bySManualyTargetPowerUV1_8 := fbAlfen8.stDataECS.bySManualyTargetPower;	
		byErrorWarningUV1_8 := fbAlfen8.stDataECS.byErrorWarning;
			rChargingTimeInMinUV1_8 := fbAlfen8.stDataECS.arrChargingTimeInMin[1];
				lrPowerUV1_8 := fbAlfen8.stDataECS.lrTotalPower;	
					wStateUV1_8 := fbAlfen8.stDataECS.arrSocketStateECS[1];
						lrEnergySessionUV1_8 := fbAlfen8.stDataECS.arrSocketEnergySession[1];
							lrTotalEnergyUV1_8 := fbAlfen8.stDataECS.lrTotalCounterEnergy_Consumption;
	
(*---------------------------------------------CS9-----------------------------------------------------------*)	
	
//Manual Power
fbAlfen9.stSetupECS.bManualyOn := bManualyOnUV1_9;
	fbAlfen9.stSetupECS.byManualyTargetPower := byManualyTargetPowerUV1_9;
	
fbAlfen9(
	bEnable:= , 
	bPowerDataInvers:= , 
	byElectricFuseLine:= , 
	byUnitID_Socket1:= 1, 
	byUnitID_Socket2:= , 
	byNumberOfSockets:= 1, 
	byNumberOfConnectionWire:= 1, 
	diNrOfEMS_IN:= prgEMS.fbEMS.diNrOfEMS_OUT, 
	diNrOfEM_IN_CS:= , 
	sIPAdress:= '192.168.1.165',  
	stSetupECS:= , 
	stDataECS=> , 
	diNrOfECS_OUT=> );

bSManualyOn_UV1_9 := fbAlfen9.stDataECS.bSManualyOn;
	bySManualyTargetPowerUV1_9 := fbAlfen9.stDataECS.bySManualyTargetPower;
		byErrorWarningUV1_9 := fbAlfen9.stDataECS.byErrorWarning;	
			rChargingTimeInMinUV1_9 := fbAlfen9.stDataECS.arrChargingTimeInMin[1];
				lrPowerUV1_9 := fbAlfen9.stDataECS.lrTotalPower;	
					wStateUV1_9 := fbAlfen9.stDataECS.arrSocketStateECS[1];
						lrEnergySessionUV1_9 := fbAlfen9.stDataECS.arrSocketEnergySession[1];
							lrTotalEnergyUV1_9 := fbAlfen9.stDataECS.lrTotalCounterEnergy_Consumption;
	
(*---------------------------------------------CS10-----------------------------------------------------------*)	
	
//Manual Power
fbAlfen10.stSetupECS.bManualyOn := bManualyOnUV1_10;
	fbAlfen10.stSetupECS.byManualyTargetPower := byManualyTargetPowerUV1_10;
	
fbAlfen10(
	bEnable:= , 
	bPowerDataInvers:= , 
	byElectricFuseLine:= , 
	byUnitID_Socket1:= 1, 
	byUnitID_Socket2:= , 
	byNumberOfSockets:= 1, 
	byNumberOfConnectionWire:= 1, 
	diNrOfEMS_IN:= prgEMS.fbEMS.diNrOfEMS_OUT, 
	diNrOfEM_IN_CS:= , 
	sIPAdress:= '192.168.1.176', 
	stSetupECS:= , 
	stDataECS=> , 
	diNrOfECS_OUT=> );

bSManualyOn_UV1_10 := fbAlfen10.stDataECS.bSManualyOn;
	bySManualyTargetPowerUV1_10 := fbAlfen10.stDataECS.bySManualyTargetPower;
		byErrorWarningUV1_10 := fbAlfen10.stDataECS.byErrorWarning;	
			rChargingTimeInMinUV1_10 := fbAlfen10.stDataECS.arrChargingTimeInMin[1];
				lrPowerUV1_10 := fbAlfen10.stDataECS.lrTotalPower;	
					wStateUV1_10 := fbAlfen10.stDataECS.arrSocketStateECS[1];
						lrEnergySessionUV1_10 := fbAlfen10.stDataECS.arrSocketEnergySession[1];
							lrTotalEnergyUV1_10 := fbAlfen10.stDataECS.lrTotalCounterEnergy_Consumption;

(*---------------------------------------------DC1-----------------------------------------------------------*)	
	
//Manual Power
fbApliT_1.stSetupECS.bManualyOn := bManualyOnDC_1;
	fbApliT_1.stSetupECS.byManualyTargetPower := byManualyTargetPowerDC_1;
	
fbApliT_1(
	bEnable:= , 
	bPowerDataInvers:= , 
	byElectricFuseLine:= , 
	byUnitID:= 1, 
	diNrOfEMS_IN:= prgEMS.fbEMS.diNrOfEMS_OUT, 
	diNrOfEM_IN_CS:= , 
	sIPAdress:= '192.168.1.177', 
	stSetupECS:= , 
	stDataECS=> , 
	diNrOfECS_OUT=> );

bSManualyOn_DC_1 := fbApliT_1.stDataECS.bSManualyOn;
	bySManualyTargetPowerDC_1 := fbApliT_1.stDataECS.bySManualyTargetPower;
		byErrorWarningDC_1 := fbApliT_1.stDataECS.byErrorWarning;
			lrPowerTotalDC1 := fbApliT_1.stDataECS.lrTotalPower;
				lrPowerDC1_S1 :=  fbApliT_1.stDataECS.arrSocketPower[1];
					lrPowerDC1_S2 :=  fbApliT_1.stDataECS.arrSocketPower[2];	 	
						rChargingTimeInMinDC1_S1 := fbApliT_1.stDataECS.arrChargingTimeInMin[1];	
							rChargingTimeInMinDC1_S2 := fbApliT_1.stDataECS.arrChargingTimeInMin[2];
								dwSOCCarDC1_S1 := fbApliT_1.stDataECS.arrSocketSOCCar[1]; 
									dwSOCCarDC1_S2 := fbApliT_1.stDataECS.arrSocketSOCCar[2]; 	
										wStateDC1_S1 := fbApliT_1.stDataECS.arrSocketStateECS[1];
											wStateDC1_S2 := fbApliT_1.stDataECS.arrSocketStateECS[2];
												lrEnergySessionDC1_S1 := fbApliT_1.stDataECS.arrSocketEnergySession[1];
													lrEnergySessionDC1_S2 := fbApliT_1.stDataECS.arrSocketEnergySession[2];
														lrTotalEnergyDC1 := fbApliT_1.stDataECS.lrTotalCounterEnergy_Consumption;			
		
(*---------------------------------------------DC2-----------------------------------------------------------*)	
	
//Manual Power
fbApliT_2.stSetupECS.bManualyOn := bManualyOnDC_2;
	fbApliT_2.stSetupECS.byManualyTargetPower := byManualyTargetPowerDC_2;
	
fbApliT_2(
	bEnable:= , 
	bPowerDataInvers:= , 
	byElectricFuseLine:= , 
	byUnitID:= 1, 
	diNrOfEMS_IN:= prgEMS.fbEMS.diNrOfEMS_OUT, 
	diNrOfEM_IN_CS:= , 
	sIPAdress:= '192.168.1.185', 
	stSetupECS:= , 
	stDataECS=> , 
	diNrOfECS_OUT=> );
	
bSManualyOn_DC_2 := fbApliT_2.stDataECS.bSManualyOn;
	bySManualyTargetPowerDC_2 := fbApliT_2.stDataECS.bySManualyTargetPower;
		byErrorWarningDC_2 := fbApliT_2.stDataECS.byErrorWarning;
			lrPowerTotalDC2 := fbApliT_2.stDataECS.lrTotalPower;
				lrPowerDC2_S1 :=  fbApliT_2.stDataECS.arrSocketPower[1];
					lrPowerDC2_S2 :=  fbApliT_2.stDataECS.arrSocketPower[2];	 	
						rChargingTimeInMinDC2_S1 := fbApliT_2.stDataECS.arrChargingTimeInMin[1];	
							rChargingTimeInMinDC2_S2 := fbApliT_2.stDataECS.arrChargingTimeInMin[2];
								dwSOCCarDC2_S1 := fbApliT_2.stDataECS.arrSocketSOCCar[1]; 
									dwSOCCarDC2_S2 := fbApliT_2.stDataECS.arrSocketSOCCar[2]; 	
										wStateDC2_S1 := fbApliT_2.stDataECS.arrSocketStateECS[1];
											wStateDC2_S2 := fbApliT_2.stDataECS.arrSocketStateECS[2];
												lrEnergySessionDC2_S1 := fbApliT_2.stDataECS.arrSocketEnergySession[1];
													lrEnergySessionDC2_S2 := fbApliT_2.stDataECS.arrSocketEnergySession[2];
														lrTotalEnergyDC2 := fbApliT_2.stDataECS.lrTotalCounterEnergy_Consumption;

END_PROGRAM

// ---- DUTs/FB_ECS_Alfen_NG9xx_Platform.TcPOU
FUNCTION_BLOCK FB_ECS_Alfen_NG9xx_Platform
VAR_INPUT PERSISTENT
	bEnable										: BOOL;																			//{#lynus.ag#()} //Enable the Fuctionblock and his logic
	bPowerDataInvers							: BOOL;																			//With True its possible to invert all received power data from the electric meter
	byElectricFuseLine							: BYTE; 																		//Electric Fuse Line on wich the ECS is connected => 1 2 3 (If 0 then this charging station is not connected to a Electric Fuse Line)
	byUnitID_Socket1							: BYTE;																			//Unit ID for Socket 1
	byUnitID_Socket2							: BYTE;																			//Unit ID for Socket 2
	byNumberOfSockets							: BYTE;																			//Give information about the number of sockets. (max 2,  min 1)
	byNumberOfConnectionWire					: BYTE;																			//Give a information about the Number of Connection Wires to the charging station. (max 2,  min 1)
	diNrOfEMS_IN								: DINT;																			//Number of EMS what control this Device.
	diNrOfEM_IN_CS								: DINT;																			//Number of the electric meter for incoming power data. (Power Data for this Device)
	sIPAdress									: STRING(15);																	//IP Adress from the Alfen charging station
	stSetupECS									: ST_Setup_ECS;																	//{#lynus.ag#()} //Setup charging station
END_VAR
VAR_OUTPUT
	stDataECS									: ST_ECS_Output;																//{#lynus.ag#()} //Electric charging station output data
	diNrOfECS_OUT								: DINT;																			//Active Number from the Electric charging Function for using on other functions
	lrTotalPowerECSRealTime						: LREAL;																		//Total Electric Power in kW read out directly from the Charging station. (Real time)
END_VAR
VAR
	{attribute 'hide'}
	fbCS										: FB_ElectricChargingStation;													//Function block for electric charging station
	{attribute 'hide'}
	fbNumberDevice								: FB_NumberOfDevice;															//Function block to calcualte the number of the Device
	fbDIExternalLock							: FB_XL1XXX_DI;																	//Digital Input from external loock signal
	
	fbMBRead_FC3								: FB_MBReadRegs;																//Modbus Read Function (FC3)
	
	fbMBWrite_FC16								: FB_MBWriteRegs;																//Modbus Write Function (FC16)
	{attribute 'hide'}
	fbConvertWordToByte							: FB_CV_WORD_TO_BYTE;															//Convert Word To Byte
	{attribute 'hide'}
	fbConvertDwordToWord						: FB_CV_DWORD_TO_WORD;															//Convert Dword to Word
	{attribute 'hide'}
	fbConvertWordToDword						: FB_CV_WORD_TO_DWORD;															//Convert Word to Dword
	{attribute 'hide'}
	fbConvertWordToUlint						: FB_CV_WORD_TO_ULINT;															//Convert Word to ULINT
	{attribute 'hide'}
	timDelay									: TON;																			//Timer for Delay between Requests
	{attribute 'hide'}
	timTimeout									: TON;																			//Timer for Timeout
	{attribute 'hide'}
	timDissableFunctions						: TON;																			//Timer to dissable the Function after Lynus_Standards.Constants_General.tTimeDissableLynusFunctions Days without connection to the Lynus Cloud
	{attribute 'hide'}
	timResetConnectionOnGVL						: TON;																			//Timer to try reset the connection Flag on the GVL. (When somebody delete the Connection Function and make only a onlinechange)
	{attribute 'hide'}
	timChTimeSocket1							: TON;																			//Charging Time for socket 1
	{attribute 'hide'}
	timChTimeSocket2							: TON;																			//Charging Time for socket 2
	{attribute 'hide'}
	timDelayStart								: TON;																			//Timer to start the state machine with Daley after enabling or after the system ist restartet
	{attribute 'hide'}
	FPError_FC_3								: R_TRIG;																		//Internal positive Edge
	{attribute 'hide'}
	FPError_FC_16								: R_TRIG;																		//Internal positive Edge
	{attribute 'hide'}
	FPEnable									: R_TRIG;																		//Internal positive Edge
	{attribute 'hide'}
	stConvertFloat								: ST_UN_FLOAT_CONVERT_DWORD_REAL;												//Convert float
	{attribute 'hide'}
	stConvertFloat2								: ST_UN_FLOAT_CONVERT_ULINT_LREAL;												//Convert float
	{attribute 'hide'}
	arrPD										: ARRAY[1..18] OF FB_PersistentData_Number;										//Function to save persistent data
	{attribute 'hide'}
	fbPDString									: FB_PersistentData_String;														//Function to save persistent string data
	{attribute 'hide'}
	arrBuffer_FC3								: ARRAY[1..5] OF WORD;															//Buffer with Data from FC3
	{attribute 'hide'}
	arrBuffer_FC16								: ARRAY[1..2] OF WORD;															//Buffer with Data from FC16
	{attribute 'hide'}
	arrMode3State								: ARRAY[1..2] OF STRING(2);														//Mode 3 State
	{attribute 'hide'}
	bErrorCS									: BOOL;																			//Error State from the charging station
	{attribute 'hide'}
	bMBTCPError									: BOOL;																			//Modbus TCP Function Error
	{attribute 'hide'}
	bySocketInProgress							: BYTE;																			//Shows the Socket in Progress when we have more then 1 Socket																		
	{attribute 'hide'}
	byWaitInStep								: BYTE;																			//Wait in Step before start to clean data on PLC
	{attribute 'hide'}
	iStateGVLData								: INT;																			//State machine to handle the data on the GVL
	{attribute 'hide'}
	iStateModbusRead							: INT;																			//State machine for read out Data over Modbus RTU
	{attribute 'hide'}
	iStateModbusWrite							: INT;																			//State machine for write Data over Modbus RTU
	{attribute 'hide'}
	iStateModbusError							: INT;																			//State machine for error out Data over Modbus RTU	
	{attribute 'hide'}
	iStateModbus_CP								: INT;																			//Variable to compare the state machine variable to set or reset the timeout timer
	{attribute 'hide'}
	diNumberOfActiveBatterys					: DINT;																			//Number of active batterys
	{attribute 'hide'}
	diNumberOfBatteryInverterInEPO				: DINT;																			//Number of battery inverters that work in Emergency Power operation 
	{attribute 'hide'}
	diLPForGVL									: DINT;																			//Loop to clean old data on GVL
	{attribute 'hide'}
	diCounterForGVL								: DINT;																			//Counter to clean old data on GVL
	{attribute 'hide'}
	dwSumSOC									: DWORD;																		//Sum of the SOC from all batterys
	{attribute 'hide'}
	lrTotalCounterEnergy_Consumption_S1			: LREAL;																		//Energy Counter Consumption in Wh Socket 1
	{attribute 'hide'}
	lrTotalCounterEnergy_Consumption_S2			: LREAL;																		//Energy Counter Consumption in Wh Socket 2
	{attribute 'hide'}
	lrTotalCounterEnergy_Production_S1			: LREAL;																		//Energy Counter Production in Wh Socket 1
	{attribute 'hide'}
	lrTotalCounterEnergy_Production_S2			: LREAL;																		//Energy Counter Production in Wh Socket 2
	{attribute 'hide'}
	rPowerECS_S1								: REAL;																			//Power from the ECS in W Socket 1
	{attribute 'hide'}
	rPowerECS_S2								: REAL;																			//Power from the ECS in W Socket 2
	{attribute 'hide'}	
	liLPBatteryData								: LINT;																			//Loop to check some data from batterys
	{attribute 'hide'}
	liLPInEPO									: LINT;																			//Loop to check if 1 or more battery inverters build a island grid
END_VAR
VAR PERSISTENT
	{attribute 'conditionalshow'}
	diNrOfEMS_IN_CP								: DINT;																			//Number of EMS what control this Device to compare with the original
END_VAR

//Creator : Kai Ebensperger
//Company : Lynus AG
//Date : 04.10.2021
//Version : 1.0.0.0

//With this Funcition its possible to communicate with a Alfen Electric charging station from the NG9xx Platform over Modbus TCP.
//Its possible to controll the charging station over the charg current
//When the Function send 0 Ampere is switched of, then the charging station is blocked and its not possible to charge
//This Function Block supports Charging stations with maximal 2 sockets
//This function controll to the charging station with 2 sockets the current / 2
//When we have 2 Connection Wires and 2 sockets on the charging station, than the function send the full current. Attention : Then on the max Power must be Insert the maxpower in kW * 2

//Versions that are supported : 2.3 Date : 30.10.2020

//NOTE for diNr.....Designation => 
//_IN = Here Data come in from other Functions or go out to other functions about the GVL
//_OUT = Here Data go out to other functions about the GVL

(*--------------------------------------------------------------------------------------------Limits-------------------------------------------------------------------------------------*)

byNumberOfSockets := LIMIT(1,byNumberOfSockets,2);
	byNumberOfConnectionWire := LIMIT(1,byNumberOfConnectionWire,2);
		diNrOfEMS_IN := LIMIT(0,diNrOfEMS_IN,Constants_Energy.diMaxNumberOfEMS);
			diNrOfEM_IN_CS := LIMIT(0,diNrOfEM_IN_CS,Constants_Energy.diMaxNumberOfElectricMeters);
				byUnitID_Socket1 := LIMIT(1,byUnitID_Socket1,1);
					byUnitID_Socket2 := LIMIT(2,byUnitID_Socket2,2);
						byElectricFuseLine := LIMIT(0,byElectricFuseLine,30);

(*------------------------------------------------------------------Power Data----------------------------------------------------------------------------*)

IF diNrOfEM_IN_CS <> 0 THEN
	//Energy Session Input data
	fbCS.bCalculateEnergySession := FALSE;
	fbCS.arrSocketPowerECS[1] := 0;
	fbCS.arrSocketPowerECS[2] := 0;
	fbCS.arrSocketPowerECS[3] := 0;
	fbCS.arrSocketPowerECS[4] := 0;
	fbCS.arrSocketEnergySession[1] := 0;
	fbCS.arrSocketEnergySession[2] := 0;
	fbCS.arrSocketEnergySession[3] := 0;
	fbCS.arrSocketEnergySession[4] := 0;
		IF NOT bPowerDataInvers THEN
			//Energy meter input data for cs Function block
			fbCS.lrCounterEnergyT1_Consumption := Lynus_Standards.GVL_Energy.stDataElectricMeters[diNrOfEM_IN_CS].lrCounterEnergyT1_Production * 1000;
			fbCS.lrCounterEnergyT2_Consumption := Lynus_Standards.GVL_Energy.stDataElectricMeters[diNrOfEM_IN_CS].lrCounterEnergyT2_Production * 1000;
			fbCS.lrCounterEnergyT1_Production := Lynus_Standards.GVL_Energy.stDataElectricMeters[diNrOfEM_IN_CS].lrCounterEnergyT1_Consumption * 1000;
			fbCS.lrCounterEnergyT2_Production := Lynus_Standards.GVL_Energy.stDataElectricMeters[diNrOfEM_IN_CS].lrCounterEnergyT1_Consumption * 1000;
			fbCS.lrTotalCounterEnergy_Consumption := Lynus_Standards.GVL_Energy.stDataElectricMeters[diNrOfEM_IN_CS].lrTotalCounterEnergy_Production * 1000;
			fbCS.lrTotalCounterEnergy_Production := Lynus_Standards.GVL_Energy.stDataElectricMeters[diNrOfEM_IN_CS].lrTotalCounterEnergy_Consumption * 1000;
				fbCS.lrTotalPowerECS := (Lynus_Standards.GVL_Energy.stDataElectricMeters[diNrOfEM_IN_CS].lrPower * 1000) * - 1;
			ELSE
			//Energy meter input data for cs Function block
			fbCS.lrCounterEnergyT1_Consumption := Lynus_Standards.GVL_Energy.stDataElectricMeters[diNrOfEM_IN_CS].lrCounterEnergyT1_Consumption * 1000;
			fbCS.lrCounterEnergyT2_Consumption := Lynus_Standards.GVL_Energy.stDataElectricMeters[diNrOfEM_IN_CS].lrCounterEnergyT2_Consumption * 1000;
			fbCS.lrCounterEnergyT1_Production := Lynus_Standards.GVL_Energy.stDataElectricMeters[diNrOfEM_IN_CS].lrCounterEnergyT1_Production * 1000;
			fbCS.lrCounterEnergyT2_Production := Lynus_Standards.GVL_Energy.stDataElectricMeters[diNrOfEM_IN_CS].lrCounterEnergyT2_Production * 1000;
			fbCS.lrTotalCounterEnergy_Consumption := Lynus_Standards.GVL_Energy.stDataElectricMeters[diNrOfEM_IN_CS].lrTotalCounterEnergy_Consumption * 1000;
			fbCS.lrTotalCounterEnergy_Production := Lynus_Standards.GVL_Energy.stDataElectricMeters[diNrOfEM_IN_CS].lrTotalCounterEnergy_Production * 1000;
				fbCS.lrTotalPowerECS := Lynus_Standards.GVL_Energy.stDataElectricMeters[diNrOfEM_IN_CS].lrPower * 1000;
		END_IF
ELSE
	//Energy meter input data for cs Function block
	fbCS.lrCounterEnergyT1_Consumption := lrTotalCounterEnergy_Consumption_S1 + lrTotalCounterEnergy_Consumption_S2;
	fbCS.lrCounterEnergyT2_Consumption := 0;
	fbCS.lrCounterEnergyT1_Production := lrTotalCounterEnergy_Production_S1 + lrTotalCounterEnergy_Production_S2;
	fbCS.lrCounterEnergyT2_Production := 0;
	fbCS.lrTotalCounterEnergy_Consumption := lrTotalCounterEnergy_Consumption_S1 + lrTotalCounterEnergy_Consumption_S2;
	fbCS.lrTotalCounterEnergy_Production := lrTotalCounterEnergy_Production_S1 + lrTotalCounterEnergy_Production_S2;
		fbCS.lrTotalPowerECS := rPowerECS_S1 + rPowerECS_S2;
	//Energy Session Input data
	fbCS.bCalculateEnergySession := TRUE;
	fbCS.arrSocketPowerECS[1] := rPowerECS_S1;
	fbCS.arrSocketPowerECS[2] := rPowerECS_S2;
	fbCS.arrSocketPowerECS[3] := 0;
	fbCS.arrSocketPowerECS[4] := 0;
	fbCS.arrSocketEnergySession[1] := lrTotalCounterEnergy_Consumption_S1;
	fbCS.arrSocketEnergySession[2] := lrTotalCounterEnergy_Consumption_S2;
	fbCS.arrSocketEnergySession[3] := 0;
	fbCS.arrSocketEnergySession[4] := 0;
END_IF			

(*-------------------------------------------------------------Calcualte the number of ECS---------------------------------------------------------------*)

fbNumberDevice(
	diActualNumberOfDevices:= Lynus_Standards.GVL_Energy.stNumberOfDevices.diNumberOfECS, 
	diMaxNumberOfDevices:= Constants_Energy.diMaxNumberOfElectricChargingStations, 
	udiCounterOnlineChange:= TwinCAT_SystemInfoVarList._AppInfo.OnlineChangeCnt, 
	bNumberIsCalculatet=> , 
	bFPNumberIsCalculatet=> , 
	bOnlineChange=> , 
	diNumberForThisDevice=> diNrOfECS_OUT, 
	diNumberOfTotalDevices=> );

//Write new Numer on GVL
IF fbNumberDevice.bFPNumberIsCalculatet THEN
	Lynus_Standards.GVL_Energy.stNumberOfDevices.diNumberOfECS := fbNumberDevice.diNumberOfTotalDevices;	
END_IF 

//Delete old Number on GVL
IF fbNumberDevice.bOnlineChange THEN 
	Lynus_Standards.GVL_Energy.stNumberOfDevices.diNumberOfECS := diNrOfECS_OUT;	
		iStateGVLData := 1;
END_IF

(*-------------------------------------------------------------Service from Backend is ready and check the connection to backen for dissabel/enable Function---------------------------------------------------------------*)

//Try to reset the variable for connection on the GVL. When all is normal then the Lynus Mqtt connection function set this variable to true in the next cycle
//When we have no connection to the backend then after Lynus_Standards.Constants_General.tTimeDissableLynusFunctions days the Function is dissabled with all of his functionalities
timResetConnectionOnGVL(IN:= NOT timResetConnectionOnGVL.Q, PT:= T#1H, Q=> , ET=> );
	IF timResetConnectionOnGVL.Q THEN Lynus_Standards.GVL_Communicator.bStateConnectionToEnableFunctions := FALSE; END_IF
		IF NOT Lynus_Standards.GVL_Communicator.bStateConnectionToEnableFunctions THEN timDissableFunctions.IN := TRUE; ELSE timDissableFunctions.IN := FALSE; END_IF  
			timDissableFunctions(IN:= , PT:= Lynus_Standards.Constants_General.tTimeDissableLynusFunctions, Q=> , ET=> );
			
(*--------------------------------------------------------------------------------------------State Machine Read--------------------------------------------------------------------------------------*)

//Timer for Delay
timDelay(IN:= , PT:= T#400MS, Q=> , ET=> );

//Timer for Timeout in Statemachine
IF (iStateModbusRead > 0 AND iStateModbusRead <= 5 AND iStateModbusRead = iStateModbus_CP) OR
		(iStateModbusWrite > 0 AND iStateModbusWrite <= 1 AND iStateModbusWrite = iStateModbus_CP) THEN
			timTimeout.IN := TRUE;
ELSE	
			timTimeout.IN := FALSE;
END_IF
	//Timeout Timer is dissabled when the Init Step is aktiv or the function is not enabled
	IF (iStateModbusRead = 0 AND iStateModbusWrite = 0) OR NOT bEnable THEN timTimeout.IN := FALSE; END_IF
		timTimeout(IN:= , PT:= T#10S, Q=> , ET=> );

//Enable with Delay that not all sockets have to be created at the same time
timDelayStart(IN:= bEnable, PT:= T#20MS * diNrOfECS_OUT, Q=> , ET=> );
	FPEnable(CLK:= timDelayStart.Q, Q=> );

IF FPEnable.Q AND iStateModbusRead = 0 AND iStateModbusWrite = 0 THEN iStateModbusRead := 1; bySocketInProgress := 1; END_IF		
		
//Not Enabled
IF NOT bEnable THEN iStateModbusRead := 0; iStateModbusError := 0; iStateModbusWrite := 0; END_IF		
		
CASE iStateModbusRead OF

	0://Init Step 
		iStateModbus_CP := 0;
			timDelay.IN := FALSE;
				fbMBRead_FC3.bExecute := FALSE;
					fbMBWrite_FC16.bExecute := FALSE;
						bySocketInProgress := 0;
							rPowerECS_S1 := 0;	
								rPowerECS_S2 := 0;	
		arrMode3State[1] := ''; arrMode3State[2] := '';
	
	1://Read Out the mode 3 State from the charging station (Register 1201)
		iStateModbus_CP := iStateModbusRead;
		
		//Reset Write
		fbMBWrite_FC16.bExecute := FALSE;
			
		//Start Read
		fbMBRead_FC3.nQuantity := 5;
			fbMBRead_FC3.nMBAddr := 1201;
				fbMBRead_FC3.bExecute := TRUE;
					IF bySocketInProgress = 1 THEN fbMBRead_FC3.nUnitID := byUnitID_Socket1;
					ELSIF bySocketInProgress = 2 THEN fbMBRead_FC3.nUnitID := byUnitID_Socket2; 
					END_IF
			
		IF fbMBRead_FC3.bBusy THEN timDelay.IN := TRUE; END_IF
		
		//Wait for Delay, copy Data and then next step
		IF NOT fbMBRead_FC3.bBusy AND NOT fbMBRead_FC3.bError AND timDelay.Q THEN
			//Mode 3 state
			fbConvertWordToByte(wInputValue:= arrBuffer_FC3[1], eByteOrderForConvert:= eByteOrder.eBigEndian, byOutputValue_1=> , byOutputValue_2=> );	
				bySocketInProgress := LIMIT(1,bySocketInProgress,2);
					IF fbConvertWordToByte.byOutputValue_1 = 16#41 AND fbConvertWordToByte.byOutputValue_2 = 16#00 THEN arrMode3State[bySocketInProgress] := 'A';
					ELSIF fbConvertWordToByte.byOutputValue_1 = 16#42 AND fbConvertWordToByte.byOutputValue_2 = 16#31 THEN arrMode3State[bySocketInProgress] := 'B1';
					ELSIF fbConvertWordToByte.byOutputValue_1 = 16#42 AND fbConvertWordToByte.byOutputValue_2 = 16#32 THEN arrMode3State[bySocketInProgress] := 'B2';  			
					ELSIF fbConvertWordToByte.byOutputValue_1 = 16#43 AND fbConvertWordToByte.byOutputValue_2 = 16#31 THEN arrMode3State[bySocketInProgress] := 'C1';
					ELSIF fbConvertWordToByte.byOutputValue_1 = 16#43 AND fbConvertWordToByte.byOutputValue_2 = 16#32 THEN arrMode3State[bySocketInProgress] := 'C2';
					ELSIF fbConvertWordToByte.byOutputValue_1 = 16#44 AND fbConvertWordToByte.byOutputValue_2 = 16#31 THEN arrMode3State[bySocketInProgress] := 'D1';
					ELSIF fbConvertWordToByte.byOutputValue_1 = 16#44 AND fbConvertWordToByte.byOutputValue_2 = 16#32 THEN arrMode3State[bySocketInProgress] := 'D2';
					ELSIF fbConvertWordToByte.byOutputValue_1 = 16#45 AND fbConvertWordToByte.byOutputValue_2 = 16#00 THEN arrMode3State[bySocketInProgress] := 'E';
					ELSIF fbConvertWordToByte.byOutputValue_1 = 16#46 AND fbConvertWordToByte.byOutputValue_2 = 16#00 THEN arrMode3State[bySocketInProgress] := 'F';
					END_IF
			//Go to Next Step
			fbMBRead_FC3.bExecute := FALSE;
				timDelay.IN := FALSE;		
					iStateModbusRead := 2;
		END_IF	

		//Error or Timeout
		IF FPError_FC_3.Q OR timTimeout.Q THEN
			iStateModbusError := 300;
		END_IF
		
	2://Power Data in W (Register 344)
		iStateModbus_CP := iStateModbusRead;

		//Start Read
		fbMBRead_FC3.nQuantity := 2;
			fbMBRead_FC3.nMBAddr := 344;
				fbMBRead_FC3.bExecute := TRUE;
					IF bySocketInProgress = 1 THEN fbMBRead_FC3.nUnitID := byUnitID_Socket1;
					ELSIF bySocketInProgress = 2 THEN fbMBRead_FC3.nUnitID := byUnitID_Socket2; 
					END_IF
			
		IF fbMBRead_FC3.bBusy THEN timDelay.IN := TRUE; END_IF
		
		//Wait for Delay, copy Data and then next step
		IF NOT fbMBRead_FC3.bBusy AND NOT fbMBRead_FC3.bError AND timDelay.Q THEN
			//Power Data in kW
			fbConvertWordToDword(wInputValue_1:= arrBuffer_FC3[1], wInputValue_2:= arrBuffer_FC3[2], eByteOrderForConvert:= eByteOrder.eBigEndian, dwOutputValue =>);
				stConvertFloat.dwRawValue := fbConvertWordToDword.dwOutputValue;
					IF bySocketInProgress = 1 THEN 
						rPowerECS_S1 := stConvertFloat.rValueFloat;
					ELSIF bySocketInProgress = 2 THEN
						rPowerECS_S2 := stConvertFloat.rValueFloat;
					END_IF
			//Go to Next Step
			fbMBRead_FC3.bExecute := FALSE;
				timDelay.IN := FALSE;		
					iStateModbusRead := 3;
		END_IF	

		//Error or Timeout
		IF FPError_FC_3.Q OR timTimeout.Q THEN
			iStateModbusError := 300;
		END_IF
	
	3://Energy Data kWh. Delivered Sum (Register 374)
		iStateModbus_CP := iStateModbusRead;

		//Start Read
		fbMBRead_FC3.nQuantity := 4;
			fbMBRead_FC3.nMBAddr := 374;
				fbMBRead_FC3.bExecute := TRUE;
					IF bySocketInProgress = 1 THEN fbMBRead_FC3.nUnitID := byUnitID_Socket1;
					ELSIF bySocketInProgress = 2 THEN fbMBRead_FC3.nUnitID := byUnitID_Socket2; 
					END_IF
			
		IF fbMBRead_FC3.bBusy THEN timDelay.IN := TRUE; END_IF
		
		//Wait for Delay, copy Data and then next step
		IF NOT fbMBRead_FC3.bBusy AND NOT fbMBRead_FC3.bError AND timDelay.Q THEN
			//Power Data in kW
			fbConvertWordToUlint(wInputValue_1:= arrBuffer_FC3[1], wInputValue_2:= arrBuffer_FC3[2], wInputValue_3:= arrBuffer_FC3[3], wInputValue_4:= arrBuffer_FC3[4], eByteOrderForConvert:= eByteOrder.eBigEndian, uliOutputValue =>);
				stConvertFloat2.uliRawValue := fbConvertWordToUlint.uliOutputValue;
					IF bySocketInProgress = 1 THEN
						lrTotalCounterEnergy_Consumption_S1 := stConvertFloat2.lrValueFloat;
					ELSIF bySocketInProgress = 2 THEN	
						lrTotalCounterEnergy_Consumption_S2 := stConvertFloat2.lrValueFloat;
					END_IF
			//Go to Next Step
			fbMBRead_FC3.bExecute := FALSE;
				timDelay.IN := FALSE;		
					iStateModbusRead := 4;
		END_IF	

		//Error or Timeout
		IF FPError_FC_3.Q OR timTimeout.Q THEN
			iStateModbusError := 300;
		END_IF
		
	4://Energy Data kWh. Consumed Sum (Register 390)
		iStateModbus_CP := iStateModbusRead;

		//Start Read
		fbMBRead_FC3.nQuantity := 4;
			fbMBRead_FC3.nMBAddr := 390;
				fbMBRead_FC3.bExecute := TRUE;
					IF bySocketInProgress = 1 THEN fbMBRead_FC3.nUnitID := byUnitID_Socket1;
					ELSIF bySocketInProgress = 2 THEN fbMBRead_FC3.nUnitID := byUnitID_Socket2; 
					END_IF
			
		IF fbMBRead_FC3.bBusy THEN timDelay.IN := TRUE; END_IF
		
		//Wait for Delay, copy Data and then next step
		IF NOT fbMBRead_FC3.bBusy AND NOT fbMBRead_FC3.bError AND timDelay.Q THEN
			//Power Data in kW
			fbConvertWordToUlint(wInputValue_1:= arrBuffer_FC3[1], wInputValue_2:= arrBuffer_FC3[2], wInputValue_3:= arrBuffer_FC3[3], wInputValue_4:= arrBuffer_FC3[4], eByteOrderForConvert:= eByteOrder.eBigEndian, uliOutputValue =>);
				stConvertFloat2.uliRawValue := fbConvertWordToUlint.uliOutputValue;
					IF bySocketInProgress = 1 THEN 
						lrTotalCounterEnergy_Production_S1 := stConvertFloat2.lrValueFloat;
					ELSIF bySocketInProgress = 2 THEN
						lrTotalCounterEnergy_Production_S2 := stConvertFloat2.lrValueFloat;
					END_IF
			//Go to Next Step
			fbMBRead_FC3.bExecute := FALSE;
				timDelay.IN := FALSE;		
					iStateModbusRead := 5;
		END_IF	

		//Error or Timeout
		IF FPError_FC_3.Q OR timTimeout.Q THEN
			iStateModbusError := 300;
		END_IF	
	
	5://Wait 1 Step to reset the delay counter befor start to write
		iStateModbus_CP := iStateModbusRead;
		
			iStateModbusWrite := 1;
				//-1 because 0 is the Init Step for Read
				iStateModbusRead := - 1;
				
			//Error on Master, changes on Inputs or Timeout
		 	IF timTimeout.Q THEN 
				iStateModbusError := 300;	 
			END_IF
	
END_CASE

//When we have only 1 connector set the mode 3 state from connector 2 to State A.
IF byNumberOfSockets = 1 THEN arrMode3State[2] := 'A'; END_IF 

(*------------------------------------------------------------------Error and Warning----------------------------------------------------------------------------*)	
 
IF arrMode3State[1] = 'F' OR arrMode3State[2] = 'F' THEN bErrorCS := TRUE; ELSE bErrorCS := FALSE; END_IF  

IF timDissableFunctions.Q THEN fbCS.bWarning := TRUE; fbCS.iWarningCode := 0; ELSE fbCS.bWarning := FALSE; END_IF   
	IF Lynus_Standards.GVL_Energy.stNumberOfDevices.diNumberOfECS > Constants_Energy.diMaxNumberOfElectricChargingStations OR bErrorCS OR bMBTCPError THEN 
		fbCS.bError := TRUE;
	ELSE 
		fbCS.bError := FALSE;
			fbCS.iErrorCode := 0;
	END_IF

IF Lynus_Standards.GVL_Energy.stNumberOfDevices.diNumberOfECS > Constants_Energy.diMaxNumberOfElectricChargingStations THEN fbCS.iErrorCode := 1;
ELSIF bErrorCS OR bMBTCPError THEN fbCS.iErrorCode := 0; END_IF

(*------------------------------------------------------------------Logic----------------------------------------------------------------------------*)

//Calcualte the total SOC if we have more then 1 battery in our system
diNumberOfActiveBatterys := 0;
	dwSumSOC := 0;
		FOR liLPBatteryData := 1 TO Constants_Energy.diMaxNumberOfBatterys BY 1 DO
			IF Lynus_Standards.GVL_Energy.stDataOfBatterys[diNrOfEMS_IN,liLPBatteryData].bEnabled THEN diNumberOfActiveBatterys := diNumberOfActiveBatterys + 1; END_IF
				dwSumSOC := dwSumSOC + Lynus_Standards.GVL_Energy.stDataOfBatterys[diNrOfEMS_IN,liLPBatteryData].dwSOC;
		END_FOR
	
IF diNumberOfActiveBatterys > 0 THEN
	fbCS.dwBatterySOC := DINT_TO_DWORD(DWORD_TO_DINT(dwSumSOC) / diNumberOfActiveBatterys);
ELSE
	fbCS.dwBatterySOC := 100;	//When we have no battery in the ems system
END_IF

//Check if one or more Batterysystems or batteryinverter make island mode
diNumberOfBatteryInverterInEPO := 0;
	FOR liLPInEPO := 1 TO Constants_Energy.diMaxNumberOfBatteryInverters BY 1 DO
		IF Lynus_Standards.GVL_Energy.stDataOfBatteryInverters[diNrOfEMS_IN,liLPInEPO].bWorkOnIslandMode THEN fbCS.bEPOIsActive := TRUE; diNumberOfBatteryInverterInEPO := diNumberOfBatteryInverterInEPO + 1; END_IF
	END_FOR 
		IF diNumberOfBatteryInverterInEPO <= 0 THEN fbCS.bEPOIsActive := FALSE; END_IF

//Digital input for external lock signal
fbDIExternalLock(bInvers:= FALSE, bSignal=> );

//Car connected to the ECS  
IF arrMode3State[1] = 'B1' OR arrMode3State[1] = 'B2' OR arrMode3State[1] = 'C1' OR arrMode3State[1] = 'C2' OR arrMode3State[1] = 'D1' OR arrMode3State[1] = 'D2' OR
	 arrMode3State[2] = 'B1' OR arrMode3State[2] = 'B2' OR arrMode3State[2] = 'C1' OR arrMode3State[2] = 'C2' OR arrMode3State[2] = 'D1' OR arrMode3State[2] = 'D2' THEN 
		fbCS.bCarConnected := TRUE; 
ELSE 
		fbCS.bCarConnected := FALSE; 
END_IF 

//Min Current
IF byNumberOfSockets <> 1 AND byNumberOfConnectionWire = 1 THEN fbCS.rMinCurrent := 12; ELSE fbCS.rMinCurrent := 6; END_IF

//Charging time
IF arrMode3State[1] = 'C2' OR arrMode3State[1] = 'D2' THEN timChTimeSocket1.IN := TRUE; ELSE timChTimeSocket1.IN := FALSE; END_IF
IF arrMode3State[2] = 'C2' OR arrMode3State[2] = 'D2' THEN timChTimeSocket2.IN := TRUE; ELSE timChTimeSocket2.IN := FALSE; END_IF  

IF timChTimeSocket1.IN THEN fbCS.arrSocketChargingTimeInput[1] := TIME_TO_REAL(timChTimeSocket1.ET) / 60000; END_IF
IF timChTimeSocket2.IN THEN fbCS.arrSocketChargingTimeInput[2] := TIME_TO_REAL(timChTimeSocket2.ET) / 60000; END_IF
fbCS.arrSocketChargingTimeInput[3] := 0;
fbCS.arrSocketChargingTimeInput[4] := 0;

timChTimeSocket1(IN:= , PT:= T#24H, Q=> , ET=> );
timChTimeSocket2(IN:= , PT:= T#24H, Q=> , ET=> );

//Mode 3 State
fbCS.arrSocketMode3StateECS[1] := arrMode3State[1];
fbCS.arrSocketMode3StateECS[2] := arrMode3State[2];
fbCS.arrSocketMode3StateECS[3] := '';
fbCS.arrSocketMode3StateECS[4] := '';

//SOC Car
fbCS.arrSOCCar[1] := 0;
fbCS.arrSOCCar[2] := 0;
fbCS.arrSOCCar[3] := 0;
fbCS.arrSOCCar[4] := 0;

//Functionblock ECS
fbCS(
	bEnable:= bEnable AND NOT timDissableFunctions.Q, 
	bError:= ,
	bWarning := ,
	bEPOIsActive:= , 
	bExternalLock:= fbDIExternalLock.bSignal, 
	bCarConnected:= , 
	bWriteWithDelay:= TRUE, 
	bCalculateEnergySession:= ,
	iErrorCode:= , 
	iWarningCode:= , 
	arrSocketChargingTimeInput:= ,
	arrSOCCar:= , 
	dwBatterySOC:= , 
	lrTotalCounterEnergy_Consumption:= , 
	lrTotalCounterEnergy_Production:= , 
	lrCounterEnergyT1_Consumption:= , 
	lrCounterEnergyT2_Consumption:= , 
	lrCounterEnergyT1_Production:= , 
	lrCounterEnergyT2_Production:= , 
	lrTotalPowerECS:= , 
	arrSocketEnergySession:= ,
	rTargetPower:= Lynus_Standards.GVL_Energy.stDataElectricChargingStations[diNrOfEMS_IN,diNrOfECS_OUT].rTargetPowerEMS, 
	rSupplyVoltage:= 692, 
	rMinCurrent:= , 
	tTimDelayOutput:= T#5S, 
	tDelayError:= T#5S,
	arrSocketMode3StateECS:= ,
	arrSocketPowerECS:= ,
	stSetupECS:= stSetupECS, 
	stDataECSOut=> , 
	stDataECSOutDelay=> stDataECS);

//Real time Power for Output
lrTotalPowerECSRealTime := fbCS.stDataECSOut.lrTotalPower;
	
(*------------------------------------------------------------------------------------------State Machine Write---------------------------------------------------------------------------------------------*)	

CASE iStateModbusWrite OF	

	1://Set the charging current (Reg 1210)
		iStateModbus_CP := iStateModbusWrite;
		
			fbMBWrite_FC16.nQuantity := 2;
				fbMBWrite_FC16.nMBAddr := 1210;
					fbMBWrite_FC16.bExecute := TRUE;
						IF bySocketInProgress = 1 THEN fbMBWrite_FC16.nUnitID := byUnitID_Socket1;
						ELSIF bySocketInProgress = 2 THEN fbMBWrite_FC16.nUnitID := byUnitID_Socket2; 
						END_IF
		
		//Prepear the sending Data. Charging Current for the charging station. (FLOAT32 format)
		//Charging current
		IF fbCS.stDataECSOut.rTargetChargeCurrent >= 0 AND fbCS.stDataECSOut.rTargetChargeCurrent <= 65535 THEN 
			IF byNumberOfSockets <> 1 AND byNumberOfConnectionWire = 1 THEN 
				stConvertFloat.rValueFloat := fbCS.stDataECSOut.rTargetChargeCurrent / 2;
			ELSE
				stConvertFloat.rValueFloat := fbCS.stDataECSOut.rTargetChargeCurrent;
			END_IF
				fbConvertDwordToWord(dwInputValue:= stConvertFloat.dwRawValue, eByteOrderForConvert:= eByteOrder.eBigEndian, wOutputValue_1=> arrBuffer_FC16[1], wOutputValue_2=> arrBuffer_FC16[2]);	 				
		END_IF	 		  
		
		IF fbMBWrite_FC16.bBusy THEN timDelay.IN := TRUE; END_IF

		//Wait for Delay and then next step
		IF NOT fbMBWrite_FC16.bBusy AND NOT fbMBWrite_FC16.bError AND timDelay.Q THEN
			fbMBWrite_FC16.bExecute := FALSE;
				timDelay.IN := FALSE;
					bMBTCPError := FALSE; 
						//Restart from new with the Read out part
						iStateModbusRead := 1;
							iStateModbusWrite := 0;
								IF byNumberOfSockets > 1 THEN 
									bySocketInProgress := bySocketInProgress + 1;
								END_IF
									IF bySocketInProgress > 2 THEN bySocketInProgress := 1; END_IF
		END_IF
				
		//Error or Timout
		IF FPError_FC_16.Q OR timTimeout.Q THEN
			iStateModbusError := 300;
		END_IF
		
END_CASE	
	
(*------------------------------------------------------------------------------------------State Machine Error---------------------------------------------------------------------------------------------*)	

CASE iStateModbusError OF
	
	300://Error
		iStateModbus_CP := iStateModbusError;
			timDelay.IN := FALSE;
				fbMBRead_FC3.bExecute := FALSE;
					fbMBWrite_FC16.bExecute := FALSE;
						bMBTCPError := TRUE; 		
							//Restart from new with the Read out part after an Error
							iStateModbusRead := 1;	
								iStateModbusError := 0;
									iStateModbusWrite := 0;
						
END_CASE

(*------------------------------------------------------------------------------------------Modbus TCP Functions---------------------------------------------------------------------------------------------*)

fbMBRead_FC3(sIPAddr:= sIPAdress, nTCPPort:= 502,cbLength:= SIZEOF(arrBuffer_FC3), pDestAddr:= ADR(arrBuffer_FC3), tTimeout:= T#5S );
	FPError_FC_3(CLK:= fbMBRead_FC3.bError, Q=> );		

fbMBWrite_FC16(sIPAddr:= sIPAdress, nTCPPort:= 502, cbLength:= SIZEOF(arrBuffer_FC16), pSrcAddr:= ADR(arrBuffer_FC16), tTimeout:= T#5S);	
	FPError_FC_16(CLK:= fbMBWrite_FC16.bError, Q=> );

(*-----------------------------------------------------------Handle data to Global structure for electric charging stations-----------------------------------------------------------------*)

//Delte al old Data on GVL after a online change or change on the variable diNrOfEMS_IDOD
IF diNrOfEMS_IN <> diNrOfEMS_IN_CP AND iStateGVLData = 0 THEN iStateGVLData := 10; END_IF 

CASE iStateGVLData OF
	
	0://Init Step
		byWaitInStep := 0;
			diCounterForGVL := 1;
	
	1://Wait for 4 Steps before clean al Data on GVL
		byWaitInStep := byWaitInStep + 1;
			IF byWaitInStep >= 4 AND fbNumberDevice.bNumberIsCalculatet THEN iStateGVLData := 2; END_IF
				//To much Devices, back to the Init step
				IF byWaitInStep >= 4 AND NOT fbNumberDevice.bNumberIsCalculatet THEN iStateGVLData := 0; END_IF	
			
	2://Clear all Data in GVL
		FOR diLPForGVL := 1 TO Constants_Energy.diMaxNumberOfEMS BY 1 DO 
			Lynus_Standards.GVL_Energy.stDataElectricChargingStations[diLPForGVL,diCounterForGVL].bEnabled := FALSE;
				Lynus_Standards.GVL_Energy.stDataElectricChargingStations[diLPForGVL,diCounterForGVL].bIsControllable := FALSE;
					Lynus_Standards.GVL_Energy.stDataElectricChargingStations[diLPForGVL,diCounterForGVL].byErrorWarning := 0;
						Lynus_Standards.GVL_Energy.stDataElectricChargingStations[diLPForGVL,diCounterForGVL].byPriority := 0;
							Lynus_Standards.GVL_Energy.stDataElectricChargingStations[diLPForGVL,diCounterForGVL].lrPower := 0;
								Lynus_Standards.GVL_Energy.stDataElectricChargingStations[diLPForGVL,diCounterForGVL].lrPowerConsumption := 0;
									Lynus_Standards.GVL_Energy.stDataElectricChargingStations[diLPForGVL,diCounterForGVL].lrPowerProduction := 0;
										Lynus_Standards.GVL_Energy.stDataElectricChargingStations[diLPForGVL,diCounterForGVL].rMaxPower := 0;
											Lynus_Standards.GVL_Energy.stDataElectricChargingStations[diLPForGVL,diCounterForGVL].byElectricFuseLine := 0;
												//Set also the target value from ems back here to 0 and not in EMS function because EMS is in Standy when we have a online change (Problem when we delete a ems function and make a online change)
												Lynus_Standards.GVL_Energy.stDataElectricChargingStations[diLPForGVL,diCounterForGVL].rTargetPowerEMS := 0;	
		END_FOR
		
			//Counter for ECS
			diCounterForGVL := diCounterForGVL + 1;
				diCounterForGVL := LIMIT(0,diCounterForGVL,Constants_Energy.diMaxNumberOfElectricChargingStations);
					//Back to the init step
					IF diCounterForGVL >= Constants_Energy.diMaxNumberOfElectricChargingStations THEN iStateGVLData := 0; END_IF

	10://Clear old Data on GVL 		
		Lynus_Standards.GVL_Energy.stDataElectricChargingStations[diNrOfEMS_IN_CP,diNrOfECS_OUT].bEnabled := FALSE;
			Lynus_Standards.GVL_Energy.stDataElectricChargingStations[diNrOfEMS_IN_CP,diNrOfECS_OUT].bIsControllable := FALSE;
				Lynus_Standards.GVL_Energy.stDataElectricChargingStations[diNrOfEMS_IN_CP,diNrOfECS_OUT].byErrorWarning := 0;
					Lynus_Standards.GVL_Energy.stDataElectricChargingStations[diNrOfEMS_IN_CP,diNrOfECS_OUT].byPriority := 0;
						Lynus_Standards.GVL_Energy.stDataElectricChargingStations[diNrOfEMS_IN_CP,diNrOfECS_OUT].lrPower := 0;
							Lynus_Standards.GVL_Energy.stDataElectricChargingStations[diNrOfEMS_IN_CP,diNrOfECS_OUT].lrPowerConsumption := 0;
								Lynus_Standards.GVL_Energy.stDataElectricChargingStations[diNrOfEMS_IN_CP,diNrOfECS_OUT].lrPowerProduction := 0;
									Lynus_Standards.GVL_Energy.stDataElectricChargingStations[diNrOfEMS_IN_CP,diNrOfECS_OUT].rMaxPower := 0;
										Lynus_Standards.GVL_Energy.stDataElectricChargingStations[diNrOfEMS_IN_CP,diNrOfECS_OUT].byElectricFuseLine := 0;
									
		diNrOfEMS_IN_CP := diNrOfEMS_IN;
			//Back to the init step
			iStateGVLData := 0;

END_CASE 	 

IF diNrOfECS_OUT > 0 AND fbNumberDevice.bNumberIsCalculatet AND diNrOfEMS_IN > 0 THEN
	Lynus_Standards.GVL_Energy.stDataElectricChargingStations[diNrOfEMS_IN,diNrOfECS_OUT].bEnabled := fbCS.stDataECSOut.bEnabled;
		Lynus_Standards.GVL_Energy.stDataElectricChargingStations[diNrOfEMS_IN,diNrOfECS_OUT].bIsControllable := TRUE;
			Lynus_Standards.GVL_Energy.stDataElectricChargingStations[diNrOfEMS_IN,diNrOfECS_OUT].byErrorWarning := fbCS.stDataECSOut.byErrorWarning;
				Lynus_Standards.GVL_Energy.stDataElectricChargingStations[diNrOfEMS_IN,diNrOfECS_OUT].byPriority := fbCS.stDataECSOut.byPriority;
					Lynus_Standards.GVL_Energy.stDataElectricChargingStations[diNrOfEMS_IN,diNrOfECS_OUT].lrPower := fbCS.stDataECSOut.lrTotalPower;
						Lynus_Standards.GVL_Energy.stDataElectricChargingStations[diNrOfEMS_IN,diNrOfECS_OUT].lrPowerConsumption := fbCS.stDataECSOut.lrTotalPowerConsumption;
							Lynus_Standards.GVL_Energy.stDataElectricChargingStations[diNrOfEMS_IN,diNrOfECS_OUT].lrPowerProduction := fbCS.stDataECSOut.lrTotalPowerProduction;
								Lynus_Standards.GVL_Energy.stDataElectricChargingStations[diNrOfEMS_IN,diNrOfECS_OUT].rMaxPower := fbCS.stDataECSOut.rMaxPower;	
									Lynus_Standards.GVL_Energy.stDataElectricChargingStations[diNrOfEMS_IN,diNrOfECS_OUT].byElectricFuseLine := byElectricFuseLine;
END_IF 

(*----------------------------------------------------------Save persistent data----------------------------------------------------------------*)

arrPD[1](lrValue:= BOOL_TO_LREAL(bEnable), bEventBasedActive=> );
arrPD[2](lrValue:= BOOL_TO_LREAL(bPowerDataInvers), bEventBasedActive=> );
arrPD[3](lrValue:= DINT_TO_LREAL(diNrOfEMS_IN), bEventBasedActive=> );
arrPD[4](lrValue:= DINT_TO_LREAL(diNrOfEM_IN_CS), bEventBasedActive=> );
arrPD[5](lrValue:= BOOL_TO_LREAL(stSetupECS.bManualyOn), bEventBasedActive=> );
arrPD[6](lrValue:= BOOL_TO_LREAL(stSetupECS.bOnEmergPowerOff), bEventBasedActive=> );
arrPD[7](lrValue:= BYTE_TO_LREAL(stSetupECS.byCSMinPower), bEventBasedActive=> );
arrPD[8](lrValue:= BYTE_TO_LREAL(stSetupECS.byDisableSOC), bEventBasedActive=> );
arrPD[9](lrValue:= BYTE_TO_LREAL(stSetupECS.byEnableSOC), bEventBasedActive=> );
arrPD[10](lrValue:= BYTE_TO_LREAL(stSetupECS.byManualyTargetPower), bEventBasedActive=> );
arrPD[11](lrValue:= BYTE_TO_LREAL(stSetupECS.byPriority), bEventBasedActive=> );
arrPD[12](lrValue:= REAL_TO_LREAL(stSetupECS.rMaxPower), bEventBasedActive=> );
arrPD[13](lrValue:= DINT_TO_LREAL(diNrOfEMS_IN_CP), bEventBasedActive=> );
arrPD[14](lrValue:= BYTE_TO_LREAL(byUnitID_Socket1), bEventBasedActive=> );
arrPD[15](lrValue:= BYTE_TO_LREAL(byUnitID_Socket2), bEventBasedActive=> );
arrPD[16](lrValue:= BYTE_TO_LREAL(byNumberOfSockets), bEventBasedActive=> );
arrPD[17](lrValue:= BYTE_TO_LREAL(byNumberOfConnectionWire), bEventBasedActive=> );
arrPD[18](lrValue:= BYTE_TO_LREAL(byElectricFuseLine), bEventBasedActive=> );
fbPDString(sText:= sIPAdress, bEventBasedActive=> );

END_FUNCTION_BLOCK

// ---- DUTs/FB_ECS_Alpitronic_Hypercharger.TcPOU
FUNCTION_BLOCK FB_ECS_Alpitronic_Hypercharger
VAR_INPUT PERSISTENT
	bEnable										: BOOL;																			//{#lynus.ag#()} //Enable the Fuctionblock and his logic
	bPowerDataInvers							: BOOL;																			//With True its possible to invert all received power data from the electric meter
	byElectricFuseLine							: BYTE; 																		//Electric Fuse Line on wich the ECS is connected => 1 2 3 (If 0 then this charging station is not connected to a Electric Fuse Line)
	byUnitID									: BYTE;																			//Unit ID 
	diNrOfEMS_IN								: DINT;																			//Number of EMS what control this Device.
	diNrOfEM_IN_CS								: DINT;																			//Number of the electric meter for incoming power data. (Power Data for this Device)
	sIPAdress									: STRING(15);																	//IP Adress from the Alfen charging station
	stSetupECS									: ST_Setup_ECS;																	//{#lynus.ag#()} //Setup charging station
END_VAR
VAR_OUTPUT
	stDataECS									: ST_ECS_Output;																//{#lynus.ag#()} //Electric charging station output data
	diNrOfECS_OUT								: DINT;																			//Active Number from the Electric charging Function for using on other functions
	lrTotalPowerECSRealTime						: LREAL;																		//Total Electric Power in kW read out directly from the Charging station. (Real time)
END_VAR
VAR
	{attribute 'hide'}
	fbCS										: FB_ElectricChargingStation;													//Function block for electric charging station
	{attribute 'hide'}
	fbNumberDevice								: FB_NumberOfDevice;															//Function block to calcualte the number of the Device
	fbDIExternalLock							: FB_XL1XXX_DI;																	//Digital Input from external loock signal
	
	fbMBRead_FC4								: FB_MBReadInputRegs ;															//Modbus Read Function (FC4)
	
	fbMBWrite_FC16								: FB_MBWriteRegs;																//Modbus Write Function (FC16)
	{attribute 'hide'}
	fbConvertDwordToWord						: FB_CV_DWORD_TO_WORD;															//Convert Dword to Word
	{attribute 'hide'}
	fbConvertWordToDord							: FB_CV_WORD_TO_DWORD;															//Convert Word to Dword
	{attribute 'hide'}
	timDelay									: TON;																			//Timer for Delay between Requests
	{attribute 'hide'}
	timTimeout									: TON;																			//Timer for Timeout
	{attribute 'hide'}
	timDissableFunctions						: TON;																			//Timer to dissable the Function after Lynus_Standards.Constants_General.tTimeDissableLynusFunctions Days without connection to the Lynus Cloud
	{attribute 'hide'}
	timResetConnectionOnGVL						: TON;																			//Timer to try reset the connection Flag on the GVL. (When somebody delete the Connection Function and make only a onlinechange)
	{attribute 'hide'}
	timDelayStart								: TON;																			//Timer to start the state machine with Daley after enabling or after the system ist restartet
	{attribute 'hide'}
	FPError_FC_4								: R_TRIG;																		//Internal positive Edge
	{attribute 'hide'}
	FPError_FC_16								: R_TRIG;																		//Internal positive Edge
	{attribute 'hide'}
	FPEnable									: R_TRIG;																		//Internal positive Edge
	{attribute 'hide'}
	arrPD										: ARRAY[1..15] OF FB_PersistentData_Number;										//Function to save persistent data
	{attribute 'conditionalshow'}
	arrEnergyCounterSocket						: ARRAY[1..4] OF FB_EnergyCounter;												//FB energy Counter, because the charging station not deliver the total energy Counter in kWh
	{attribute 'hide'}
	fbPDString									: FB_PersistentData_String;														//Function to save persistent string data
	{attribute 'hide'}
	arrBuffer_FC4								: ARRAY[1..9] OF WORD;															//Buffer with Data from FC3
	{attribute 'hide'}
	arrBuffer_FC16								: ARRAY[1..2] OF WORD;															//Buffer with Data from FC16
	{attribute 'hide'}
	arrConnectorState							: ARRAY[1..4] OF WORD;															//Connector State
	{attribute 'hide'}
	arrChargingTime								: ARRAY[1..4] OF WORD;															//Charging Time in seconds
	{attribute 'hide'}
	arrSOCCar									: ARRAY[1..4] OF WORD;															//SOC from the Car
	{attribute 'hide'}
	arrPowerConnector							: ARRAY[1..4] OF DWORD;															//Power in W from each Connector
	{attribute 'hide'}
	arrEnergySession							: ARRAY[1..4] OF REAL;															//Energy Session in kWh
	{attribute 'hide'}
	bErrorCS									: BOOL;																			//Error State from the charging station
	{attribute 'hide'}
	bMBTCPError									: BOOL;																			//Modbus TCP Function Error																	
	{attribute 'hide'}
	byWaitInStep								: BYTE;																			//Wait in Step before start to clean data on PLC
	{attribute 'hide'}
	iStateGVLData								: INT;																			//State machine to handle the data on the GVL
	{attribute 'hide'}
	iStateModbusRead							: INT;																			//State machine for read out Data over Modbus RTU
	{attribute 'hide'}
	iStateModbusWrite							: INT;																			//State machine for write Data over Modbus RTU
	{attribute 'hide'}
	iStateModbusError							: INT;																			//State machine for error out Data over Modbus RTU	
	{attribute 'hide'}
	iStateModbus_CP								: INT;																			//Variable to compare the state machine variable to set or reset the timeout timer
	{attribute 'hide'}
	wNumberOfConnectors							: WORD;																			//Number of real connecotrs on the charging station
	{attribute 'hide'}
	wStationState								: WORD;																			//Charging Station State
	{attribute 'hide'}
	wConnectorInProgress						: WORD;																			//Shows the Connector in Progress when we have more then 1 Connector	
	{attribute 'hide'}
	diNumberOfActiveBatterys					: DINT;																			//Number of active batterys
	{attribute 'hide'}
	diNumberOfBatteryInverterInEPO				: DINT;																			//Number of battery inverters that work in Emergency Power operation 
	{attribute 'hide'}
	diLPForGVL									: DINT;																			//Loop to clean old data on GVL
	{attribute 'hide'}
	diCounterForGVL								: DINT;																			//Counter to clean old data on GVL
	{attribute 'hide'}
	dwSumSOC									: DWORD;																		//Sum of the SOC from all batterys
	{attribute 'hide'}
	dwTargetPower								: DWORD;																		//Target Power in Watt to send to the charging station
	{attribute 'hide'}
	liLPBatteryData								: LINT;																			//Loop to check some data from batterys
	{attribute 'hide'}
	liLPInEPO									: LINT;																			//Loop to check if 1 or more battery inverters build a island grid
END_VAR
VAR PERSISTENT
	{attribute 'conditionalshow'}
	diNrOfEMS_IN_CP								: DINT;																			//Number of EMS what control this Device to compare with the original
END_VAR

//Creator : Kai Ebensperger
//Company : Lynus AG
//Date : 07.10.2021
//Version : 1.0.0.0

//With this Funcition its possible to communicate with a Alpitronic Hypercharger charging station over Modbus TCP.
//Its possible to controll the charging station over the charge power with the unit W
//This Charging station is a DC Hypercharger System.
//This API deliver the real Number of Connectors on the charging station
//To switch off the charging station send 0 Power to the charging station
//The minimal Curretn is set to 7.5 Ampere on AC site, bacause with al values that are < 5kW its not possible to charge the Car on DC site
//This Function Block support maximal 4 Connectors

//Versions that are supported : 1.3A Date : October 2020

//NOTE for diNr.....Designation => 
//_IN = Here Data come in from other Functions or go out to other functions about the GVL
//_OUT = Here Data go out to other functions about the GVL

(*--------------------------------------------------------------------------------------------Limits-------------------------------------------------------------------------------------*)

diNrOfEMS_IN := LIMIT(0,diNrOfEMS_IN,Constants_Energy.diMaxNumberOfEMS);
	diNrOfEM_IN_CS := LIMIT(0,diNrOfEM_IN_CS,Constants_Energy.diMaxNumberOfElectricMeters);	

(*------------------------------------------------------------------Power Data----------------------------------------------------------------------------*)

//Energy Counter Functions
arrEnergyCounterSocket[1](
	byActiveTariff:= 1, 
	lrPowerInput:= DWORD_TO_REAL(arrPowerConnector[1]) / 1000, 
	lrTotalCounterEnergy_Consumption=> , 
	lrTotalCounterEnergy_Production=> , 
	lrCounterEnergyT1_Consumption=> , 
	lrCounterEnergyT2_Consumption=> , 
	lrCounterEnergyT1_Production=> , 
	lrCounterEnergyT2_Production=> );
	
arrEnergyCounterSocket[2](
	byActiveTariff:= 1, 
	lrPowerInput:= DWORD_TO_REAL(arrPowerConnector[2]) / 1000, 
	lrTotalCounterEnergy_Consumption=> , 
	lrTotalCounterEnergy_Production=> , 
	lrCounterEnergyT1_Consumption=> , 
	lrCounterEnergyT2_Consumption=> , 
	lrCounterEnergyT1_Production=> , 
	lrCounterEnergyT2_Production=> );

arrEnergyCounterSocket[3](
	byActiveTariff:= 1, 
	lrPowerInput:= DWORD_TO_REAL(arrPowerConnector[3]) / 1000, 
	lrTotalCounterEnergy_Consumption=> , 
	lrTotalCounterEnergy_Production=> , 
	lrCounterEnergyT1_Consumption=> , 
	lrCounterEnergyT2_Consumption=> , 
	lrCounterEnergyT1_Production=> , 
	lrCounterEnergyT2_Production=> );	
	
arrEnergyCounterSocket[4](
	byActiveTariff:= 1, 
	lrPowerInput:= DWORD_TO_REAL(arrPowerConnector[4]) / 1000, 
	lrTotalCounterEnergy_Consumption=> , 
	lrTotalCounterEnergy_Production=> , 
	lrCounterEnergyT1_Consumption=> , 
	lrCounterEnergyT2_Consumption=> , 
	lrCounterEnergyT1_Production=> , 
	lrCounterEnergyT2_Production=> );

IF diNrOfEM_IN_CS <> 0 THEN
	//Energy Session Input data
	fbCS.bCalculateEnergySession := FALSE;
	fbCS.arrSocketPowerECS[1] := 0;
	fbCS.arrSocketPowerECS[2] := 0;
	fbCS.arrSocketPowerECS[3] := 0;
	fbCS.arrSocketPowerECS[4] := 0;
	fbCS.arrSocketEnergySession[1] := 0;
	fbCS.arrSocketEnergySession[2] := 0;
	fbCS.arrSocketEnergySession[3] := 0;
	fbCS.arrSocketEnergySession[4] := 0;
		IF NOT bPowerDataInvers THEN
			//Energy meter input data for cs Function block
			fbCS.lrCounterEnergyT1_Consumption := Lynus_Standards.GVL_Energy.stDataElectricMeters[diNrOfEM_IN_CS].lrCounterEnergyT1_Production * 1000;
			fbCS.lrCounterEnergyT2_Consumption := Lynus_Standards.GVL_Energy.stDataElectricMeters[diNrOfEM_IN_CS].lrCounterEnergyT2_Production * 1000;
			fbCS.lrCounterEnergyT1_Production := Lynus_Standards.GVL_Energy.stDataElectricMeters[diNrOfEM_IN_CS].lrCounterEnergyT1_Consumption * 1000;
			fbCS.lrCounterEnergyT2_Production := Lynus_Standards.GVL_Energy.stDataElectricMeters[diNrOfEM_IN_CS].lrCounterEnergyT1_Consumption * 1000;
			fbCS.lrTotalCounterEnergy_Consumption := Lynus_Standards.GVL_Energy.stDataElectricMeters[diNrOfEM_IN_CS].lrTotalCounterEnergy_Production * 1000;
			fbCS.lrTotalCounterEnergy_Production := Lynus_Standards.GVL_Energy.stDataElectricMeters[diNrOfEM_IN_CS].lrTotalCounterEnergy_Consumption * 1000;
				fbCS.lrTotalPowerECS := (Lynus_Standards.GVL_Energy.stDataElectricMeters[diNrOfEM_IN_CS].lrPower * 1000) * - 1;
		ELSE
			//Energy meter input data for cs Function block
			fbCS.lrCounterEnergyT1_Consumption := Lynus_Standards.GVL_Energy.stDataElectricMeters[diNrOfEM_IN_CS].lrCounterEnergyT1_Consumption * 1000;
			fbCS.lrCounterEnergyT2_Consumption := Lynus_Standards.GVL_Energy.stDataElectricMeters[diNrOfEM_IN_CS].lrCounterEnergyT2_Consumption * 1000;
			fbCS.lrCounterEnergyT1_Production := Lynus_Standards.GVL_Energy.stDataElectricMeters[diNrOfEM_IN_CS].lrCounterEnergyT1_Production * 1000;
			fbCS.lrCounterEnergyT2_Production := Lynus_Standards.GVL_Energy.stDataElectricMeters[diNrOfEM_IN_CS].lrCounterEnergyT2_Production * 1000;
			fbCS.lrTotalCounterEnergy_Consumption := Lynus_Standards.GVL_Energy.stDataElectricMeters[diNrOfEM_IN_CS].lrTotalCounterEnergy_Consumption * 1000;
			fbCS.lrTotalCounterEnergy_Production := Lynus_Standards.GVL_Energy.stDataElectricMeters[diNrOfEM_IN_CS].lrTotalCounterEnergy_Production * 1000;
				fbCS.lrTotalPowerECS := Lynus_Standards.GVL_Energy.stDataElectricMeters[diNrOfEM_IN_CS].lrPower * 1000;
		END_IF
ELSE
	//Energy meter input data for cs Function block
	fbCS.lrCounterEnergyT1_Consumption := arrEnergyCounterSocket[1].lrCounterEnergyT1_Consumption + arrEnergyCounterSocket[2].lrCounterEnergyT1_Consumption + arrEnergyCounterSocket[3].lrCounterEnergyT1_Consumption + arrEnergyCounterSocket[4].lrCounterEnergyT1_Consumption;
	fbCS.lrCounterEnergyT1_Consumption := fbCS.lrCounterEnergyT1_Consumption * 1000;
	fbCS.lrCounterEnergyT2_Consumption := arrEnergyCounterSocket[1].lrCounterEnergyT2_Consumption + arrEnergyCounterSocket[2].lrCounterEnergyT2_Consumption + arrEnergyCounterSocket[3].lrCounterEnergyT2_Consumption + arrEnergyCounterSocket[4].lrCounterEnergyT2_Consumption;
	fbCS.lrCounterEnergyT2_Consumption := fbCS.lrCounterEnergyT2_Consumption * 1000;
	fbCS.lrCounterEnergyT1_Production := arrEnergyCounterSocket[1].lrCounterEnergyT1_Production + arrEnergyCounterSocket[2].lrCounterEnergyT1_Production + arrEnergyCounterSocket[3].lrCounterEnergyT1_Production + arrEnergyCounterSocket[4].lrCounterEnergyT1_Production;
	fbCS.lrCounterEnergyT1_Production := fbCS.lrCounterEnergyT1_Production * 1000;
	fbCS.lrCounterEnergyT2_Production := arrEnergyCounterSocket[1].lrCounterEnergyT2_Production + arrEnergyCounterSocket[2].lrCounterEnergyT2_Production + arrEnergyCounterSocket[3].lrCounterEnergyT2_Production + arrEnergyCounterSocket[4].lrCounterEnergyT2_Production;
	fbCS.lrCounterEnergyT2_Production := fbCS.lrCounterEnergyT2_Production * 1000;
	fbCS.lrTotalCounterEnergy_Consumption := fbCS.lrCounterEnergyT1_Consumption + fbCS.lrCounterEnergyT2_Consumption;
	fbCS.lrTotalCounterEnergy_Production := fbCS.lrCounterEnergyT1_Production + fbCS.lrCounterEnergyT2_Production;
		fbCS.lrTotalPowerECS := arrPowerConnector[1] + arrPowerConnector[2] + arrPowerConnector[3] + arrPowerConnector[4];
	//Energy Session Input data
	fbCS.bCalculateEnergySession := FALSE;
	fbCS.arrSocketPowerECS[1] := arrPowerConnector[1];
	fbCS.arrSocketPowerECS[2] := arrPowerConnector[2];
	fbCS.arrSocketPowerECS[3] := arrPowerConnector[3];
	fbCS.arrSocketPowerECS[4] := arrPowerConnector[4];
	fbCS.arrSocketEnergySession[1] := arrEnergySession[1] * 1000;
	fbCS.arrSocketEnergySession[2] := arrEnergySession[2] * 1000;
	fbCS.arrSocketEnergySession[3] := arrEnergySession[3] * 1000;
	fbCS.arrSocketEnergySession[4] := arrEnergySession[4] * 1000;
END_IF			

(*-------------------------------------------------------------Calcualte the number of ECS---------------------------------------------------------------*)

fbNumberDevice(
	diActualNumberOfDevices:= Lynus_Standards.GVL_Energy.stNumberOfDevices.diNumberOfECS, 
	diMaxNumberOfDevices:= Constants_Energy.diMaxNumberOfElectricChargingStations, 
	udiCounterOnlineChange:= TwinCAT_SystemInfoVarList._AppInfo.OnlineChangeCnt, 
	bNumberIsCalculatet=> , 
	bFPNumberIsCalculatet=> , 
	bOnlineChange=> , 
	diNumberForThisDevice=> diNrOfECS_OUT, 
	diNumberOfTotalDevices=> );

//Write new Numer on GVL
IF fbNumberDevice.bFPNumberIsCalculatet THEN
	Lynus_Standards.GVL_Energy.stNumberOfDevices.diNumberOfECS := fbNumberDevice.diNumberOfTotalDevices;	
END_IF 

//Delete old Number on GVL
IF fbNumberDevice.bOnlineChange THEN 
	Lynus_Standards.GVL_Energy.stNumberOfDevices.diNumberOfECS := diNrOfECS_OUT;	
		iStateGVLData := 1;
END_IF

(*-------------------------------------------------------------Service from Backend is ready and check the connection to backen for dissabel/enable Function---------------------------------------------------------------*)

//Try to reset the variable for connection on the GVL. When all is normal then the Lynus Mqtt connection function set this variable to true in the next cycle
//When we have no connection to the backend then after Lynus_Standards.Constants_General.tTimeDissableLynusFunctions days the Function is dissabled with all of his functionalities
timResetConnectionOnGVL(IN:= NOT timResetConnectionOnGVL.Q, PT:= T#1H, Q=> , ET=> );
	IF timResetConnectionOnGVL.Q THEN Lynus_Standards.GVL_Communicator.bStateConnectionToEnableFunctions := FALSE; END_IF
		IF NOT Lynus_Standards.GVL_Communicator.bStateConnectionToEnableFunctions THEN timDissableFunctions.IN := TRUE; ELSE timDissableFunctions.IN := FALSE; END_IF  
			timDissableFunctions(IN:= , PT:= Lynus_Standards.Constants_General.tTimeDissableLynusFunctions, Q=> , ET=> );
			
(*--------------------------------------------------------------------------------------------State Machine Read--------------------------------------------------------------------------------------*)

//Timer for Delay
timDelay(IN:= , PT:= T#400MS, Q=> , ET=> );

//Timer for Timeout in Statemachine
IF (iStateModbusRead > 0 AND iStateModbusRead <= 3 AND iStateModbusRead = iStateModbus_CP) OR
		(iStateModbusWrite > 0 AND iStateModbusWrite <= 1 AND iStateModbusWrite = iStateModbus_CP) THEN
			timTimeout.IN := TRUE;
ELSE	
			timTimeout.IN := FALSE;
END_IF 
	//Timeout Timer is dissabled when the Init Step is aktiv or the function is not enabled
	IF (iStateModbusRead = 0 AND iStateModbusWrite = 0) OR NOT bEnable THEN timTimeout.IN := FALSE; END_IF
		timTimeout(IN:= , PT:= T#10S, Q=> , ET=> );

//Enable with Delay that not all sockets have to be created at the same time
timDelayStart(IN:= bEnable, PT:= T#20MS * diNrOfECS_OUT, Q=> , ET=> );
	FPEnable(CLK:= timDelayStart.Q, Q=> );

IF FPEnable.Q AND iStateModbusRead = 0 AND iStateModbusWrite = 0 THEN iStateModbusRead := 1; wConnectorInProgress := 1; END_IF		
		
//Not Enabled
IF NOT bEnable THEN iStateModbusRead := 0; iStateModbusError := 0; iStateModbusWrite := 0; END_IF		
		
CASE iStateModbusRead OF

	0://Init Step 
		iStateModbus_CP := 0;
			timDelay.IN := FALSE;
				fbMBRead_FC4.bExecute := FALSE;
					fbMBWrite_FC16.bExecute := FALSE;
						wConnectorInProgress := 0;
		arrConnectorState[1] := 0; arrConnectorState[2] := 0; arrConnectorState[3] := 0; arrConnectorState[4] := 0;
	
	1://Read Out the Number of connectors and the Charging station State (Register 2 and 3)
		iStateModbus_CP := iStateModbusRead;
		
		//Reset Write
		fbMBWrite_FC16.bExecute := FALSE;
			
		//Start Read
		fbMBRead_FC4.nQuantity := 2;
			fbMBRead_FC4.nMBAddr := 2;
				fbMBRead_FC4.bExecute := TRUE;
					fbMBRead_FC4.nUnitID := byUnitID;
			
		IF fbMBRead_FC4.bBusy THEN timDelay.IN := TRUE; END_IF
		
		//Wait for Delay, copy Data and then next step
		IF NOT fbMBRead_FC4.bBusy AND NOT fbMBRead_FC4.bError AND timDelay.Q THEN
			//Number of real Connectors
			wNumberOfConnectors := arrBuffer_FC4[1];
			//Charging station State
			wStationState := arrBuffer_FC4[2];	 
			//Connector in Progress
			wConnectorInProgress := LIMIT(1,wConnectorInProgress,4);
			//Go to Next Step
			fbMBRead_FC4.bExecute := FALSE;
				timDelay.IN := FALSE;		
					iStateModbusRead := 2;
		END_IF	

		//Error or Timeout
		IF FPError_FC_4.Q OR timTimeout.Q THEN
			iStateModbusError := 300;
		END_IF
		
	2://Read Out the Information of the real connecotrs (Register "1"00 to "1"08)
		iStateModbus_CP := iStateModbusRead;
		
		//Start Read
		fbMBRead_FC4.nQuantity := 9;
			fbMBRead_FC4.nMBAddr := 100 * wConnectorInProgress;
				fbMBRead_FC4.bExecute := TRUE;
					fbMBRead_FC4.nUnitID := byUnitID;
			
		IF fbMBRead_FC4.bBusy THEN timDelay.IN := TRUE; END_IF
		
